//motion row 3, cycle cont / single
ModeRow3	(	iStationNumber		:=1,
				iRowNumber			:=3,
				iAdvanceLimit		:=gHMIButtons.btnFdbk.btn10Fdbk,
				iReturnLimit		:=gHMIButtons.btnFdbk.btn13Fdbk,
				iAdvanceCoil		:=gModeAlternate.gModeButtons.gMotionRow3btn.btnAdvance,
				iReturnCoil			:=gModeAlternate.gModeButtons.gMotionRow3btn.btnReturn,
				iAdvanceTime		:=,
				iReturnTime			:=,
				iAdvanceInterlock	:=,
				iReturnInterlock	:=,
				iAdvancePrompt		:=,
				iReturnPrompt		:=,
				iConfig				:=RowConfig.FullRowNoVal,
				iAdvanceNumber		:=0,
				iReturnNumber		:=0,
				iUnits				:='',
				iPosn				:='',
				NumRows				:=tNumRows,
				MotionRowLocation	:=gModeAlternate.gModeRows.gMotionRow3,
				MotionRowBtnLocation:=gModeAlternate.gModeButtons.gMotionRow3btn
				);
				
//manually set row number for textlist offset				
gModeAlternate.gModeRows.gMotionRow3.IndexLocation := gModeAlternate.gModeRows.gMotionRow3.IndexLocation + 10000;			


//motion row 4, cycle start / stop
ModeRow4	(	iStationNumber		:=1,
				iRowNumber			:=4,
				iAdvanceLimit		:=gHMIButtons.btnFdbk.btnAutoCyclingFdbk,
				iReturnLimit		:=NOT gHMIButtons.btnFdbk.btnAutoCyclingFdbk,
				iAdvanceCoil		:=gModeAlternate.gModeButtons.gMotionRow4btn.btnAdvance,
				iReturnCoil			:=gModeAlternate.gModeButtons.gMotionRow4btn.btnReturn,
				iAdvanceTime		:=,
				iReturnTime			:=,
				iAdvanceInterlock	:=,
				iReturnInterlock	:=,
				iAdvancePrompt		:=,
				iReturnPrompt		:=,
				iConfig				:=RowConfig.FullRowNoVal,
				iAdvanceNumber		:=0,
				iReturnNumber		:=0,
				iUnits				:='',
				iPosn				:='',
				NumRows				:=tNumRows,
				MotionRowLocation	:=gModeAlternate.gModeRows.gMotionRow4,
				MotionRowBtnLocation:=gModeAlternate.gModeButtons.gMotionRow4btn
				);
				
//manually set row number for textlist offset				
gModeAlternate.gModeRows.gMotionRow4.IndexLocation := gModeAlternate.gModeRows.gMotionRow4.IndexLocation + 10000;			

//motion row 5, return home
ModeRow5	(	iStationNumber		:=1,
				iRowNumber			:=5,
				iAdvanceLimit		:=gHMIData.hmiHeader.homestate = 2,
				iReturnLimit		:=gHMIData.hmiHeader.homestate <> 2,
				iAdvanceCoil		:=gModeAlternate.gModeButtons.gMotionRow5btn.btnAdvance,
				iReturnCoil			:=gModeAlternate.gModeButtons.gMotionRow5btn.btnReturn,
				iAdvanceTime		:=,
				iReturnTime			:=,
				iAdvanceInterlock	:=,
				iReturnInterlock	:=,
				iAdvancePrompt		:=,
				iReturnPrompt		:=,
				iConfig				:=RowConfig.OnlyRightNoVal,
				iAdvanceNumber		:=0,
				iReturnNumber		:=0,
				iUnits				:='',
				iPosn				:='',
				NumRows				:=tNumRows,
				MotionRowLocation	:=gModeAlternate.gModeRows.gMotionRow5,
				MotionRowBtnLocation:=gModeAlternate.gModeButtons.gMotionRow5btn
				);
				
//manually set row number for textlist offset				
gModeAlternate.gModeRows.gMotionRow5.IndexLocation := gModeAlternate.gModeRows.gMotionRow5.IndexLocation + 10000;			

//motion row 6, spare
ModeRow6	(	iStationNumber		:=1,
				iRowNumber			:=6,
				iAdvanceLimit		:=FALSE,
				iReturnLimit		:=FALSE,
				iAdvanceCoil		:=gModeAlternate.gModeButtons.gMotionRow6btn.btnAdvance,
				iReturnCoil			:=gModeAlternate.gModeButtons.gMotionRow6btn.btnReturn,
				iAdvanceTime		:=,
				iReturnTime			:=,
				iAdvanceInterlock	:=,
				iReturnInterlock	:=,
				iAdvancePrompt		:=,
				iReturnPrompt		:=,
				iConfig				:=RowConfig.HideAll,
				iAdvanceNumber		:=0,
				iReturnNumber		:=0,
				iUnits				:='',
				iPosn				:='',
				NumRows				:=tNumRows,
				MotionRowLocation	:=gModeAlternate.gModeRows.gMotionRow6,
				MotionRowBtnLocation:=gModeAlternate.gModeButtons.gMotionRow6btn
				);
				
//manually set row number for textlist offset				
gModeAlternate.gModeRows.gMotionRow6.IndexLocation := gModeAlternate.gModeRows.gMotionRow6.IndexLocation + 10000;			

//motion row 7, spare
ModeRow7	(	iStationNumber		:=1,
				iRowNumber			:=7,
				iAdvanceLimit		:=FALSE,
				iReturnLimit		:=FALSE,
				iAdvanceCoil		:=gModeAlternate.gModeButtons.gMotionRow7btn.btnAdvance,
				iReturnCoil			:=gModeAlternate.gModeButtons.gMotionRow7btn.btnReturn,
				iAdvanceTime		:=,
				iReturnTime			:=,
				iAdvanceInterlock	:=,
				iReturnInterlock	:=,
				iAdvancePrompt		:=,
				iReturnPrompt		:=,
				iConfig				:=RowConfig.HideAll,
				iAdvanceNumber		:=0,
				iReturnNumber		:=0,
				iUnits				:='',
				iPosn				:='',
				NumRows				:=tNumRows,
				MotionRowLocation	:=gModeAlternate.gModeRows.gMotionRow7,
				MotionRowBtnLocation:=gModeAlternate.gModeButtons.gMotionRow7btn
				);

//manually set row number for textlist offset				
gModeAlternate.gModeRows.gMotionRow7.IndexLocation := gModeAlternate.gModeRows.gMotionRow7.IndexLocation + 10000;			
				
//motion row 8, gate lock, return only
ModeRow8	(	iStationNumber		:=1,
				iRowNumber			:=8,
				iAdvanceLimit		:=FALSE,
				iReturnLimit		:=gHMIButtons.btnFdbk.btn22Fdbk,
				iAdvanceCoil		:=gModeAlternate.gModeButtons.gMotionRow8btn.btnAdvance,
				iReturnCoil			:=gModeAlternate.gModeButtons.gMotionRow8btn.btnReturn,
				iAdvanceTime		:=,
				iReturnTime			:=,
				iAdvanceInterlock	:=,
				iReturnInterlock	:=,
				iAdvancePrompt		:=,
				iReturnPrompt		:=,
				iConfig				:=RowConfig.OnlyRightNoVal,
				iAdvanceNumber		:=0,
				iReturnNumber		:=0,
				iUnits				:='',
				iPosn				:='',
				NumRows				:=tNumRows,
				MotionRowLocation	:=gModeAlternate.gModeRows.gMotionRow8,
				MotionRowBtnLocation:=gModeAlternate.gModeButtons.gMotionRow8btn
				);
				
//manually set row number for textlist offset				
gModeAlternate.gModeRows.gMotionRow8.IndexLocation := gModeAlternate.gModeRows.gMotionRow8.IndexLocation + 10000;			

//motion row 9, gate unlocks
ModeRow9	(	iStationNumber		:=1,
				iRowNumber			:=9,
				iAdvanceLimit		:=gHMIButtons.btnFdbk.btn20Fdbk,
				iReturnLimit		:=gHMIButtons.btnFdbk.btn21Fdbk,
				iAdvanceCoil		:=gModeAlternate.gModeButtons.gMotionRow9btn.btnAdvance,
				iReturnCoil			:=gModeAlternate.gModeButtons.gMotionRow9btn.btnReturn,
				iAdvanceTime		:=,
				iReturnTime			:=,
				iAdvanceInterlock	:=,
				iReturnInterlock	:=,
				iAdvancePrompt		:=,
				iReturnPrompt		:=,
				iConfig				:=RowConfig.FullRowNoVal,
				iAdvanceNumber		:=0,
				iReturnNumber		:=0,
				iUnits				:='',
				iPosn				:='',
				NumRows				:=tNumRows,
				MotionRowLocation	:=gModeAlternate.gModeRows.gMotionRow9,
				MotionRowBtnLocation:=gModeAlternate.gModeButtons.gMotionRow9btn
				);
				
//manually set row number for textlist offset				
gModeAlternate.gModeRows.gMotionRow9.IndexLocation := gModeAlternate.gModeRows.gMotionRow9.IndexLocation + 10000;
END_ACTION

END_PROGRAM

// ---- HMI1/Screens/Machine Settings/pouMachineSettings.TcPOU
PROGRAM pouMachineSettings
VAR
	btnOSRRead:R_TRIG;
	btnOSRWrite:R_TRIG;
	ii: INT;
	OSRReadLogicDone:R_TRIG;
	
	csvRead:FB_ReadParams;
	csvWrite:FB_WriteParams;
END_VAR

//capture OSR for buttons
btnOSRRead	(	CLK := MachineSettings.btnRead);
btnOSRWrite	(	CLK := MachineSettings.btnWrite);

actReadFile();
actWriteFile();


IF MachineSettings.varSelectedRowValid THEN
		MachineSettings.numSelectedSetting := MachineSettings.Setting[MachineSettings.varSelectedRow].Value;
END_IF

IF MachineSettings.btnMoveValue THEN
	  IF 	MachineSettings.Setting[MachineSettings.varSelectedRow].Value <> MachineSettings.numSelectedSettingNew THEN
			
			//update view
			MachineSettings.Setting[MachineSettings.varSelectedRow].hasChanged := TRUE;
			MachineSettings.Setting[MachineSettings.varSelectedRow].Value := 	MachineSettings.numSelectedSettingNew;
			
			//update data area to write to
			MachineSettings.csvData[MachineSettings.varSelectedRow,1] := INT_TO_STRING (MachineSettings.Setting[MachineSettings.varSelectedRow].Value);
	  END_IF
END_IF


//feedback status
IF csvRead.qStep > 1 THEN
	MachineSettings.strStatusFeeback := 'Reading...';
END_IF
IF csvWrite.qStep > 1 THEN
	MachineSettings.strStatusFeeback := 'Writing...';
END_IF
IF csvRead.qStep = 0 AND csvWrite.qStep = 0 THEN
	MachineSettings.strStatusFeeback := '';
END_IF

IF csvRead.qErrId > 0 THEN
	MachineSettings.strStatusFeeback := CONCAT(STR1:='Read Error ',STR2:=UDINT_TO_STRING(csvRead.qErrId));
END_IF
IF csvWrite.qErrId > 0 THEN
	MachineSettings.strStatusFeeback := CONCAT(STR1:='Write Error ',STR2:=UDINT_TO_STRING(csvWrite.qErrId));
END_IF

ACTION actReadFile:
//read data
csvRead (iRead :=btnOSRRead.Q,
		iNetId :=,
		iFileName:=constCSV.str_mc_filelocation,
		iqdatabase := MachineSettings.csvData
		);

	//check state as output
	OSRReadLogicDone(clk := csvRead.qStep = 0);
	
	
//tidy up HMI screen data
IF OSRReadLogicDone.Q THEN
	MachineSettings.numElementsOfSettings := 0;
	FOR ii:=0 TO 100 DO
		MachineSettings.numElementsOfSettings := ii;
		MachineSettings.Setting[ii].Value := STRING_TO_INT(MachineSettings.csvData[ii,1]);
		MachineSettings.Setting[ii].TextName := MachineSettings.csvData[ii,0];
		MachineSettings.Setting[ii].hasChanged := FALSE;
		IF MachineSettings.csvData[ii,0] = '' THEN
			RETURN;
		END_IF
	END_FOR;
END_IF
END_ACTION

ACTION actWriteFile:
//write data
csvWrite (iWrite :=btnOSRWrite.Q,
		iNetId :=,
		iFileName:=constCSV.str_mc_filelocation,
		iqdatabase := MachineSettings.csvData
		);
		
//tidy up HMI screen data		
IF btnOSRWrite.Q THEN
	FOR ii:=0 TO 100 DO
		MachineSettings.Setting[ii].hasChanged := FALSE;
	END_FOR;
END_IF
END_ACTION

END_PROGRAM

// ---- HMI1/Screens/Machine Settings/FB_ReadParams.TcPOU
FUNCTION_BLOCK FB_ReadParams
VAR_INPUT
	iRead			: BOOL := FALSE;(* Rising edge starts program execution *)
	iNetId			: T_AmsNetId := '';	(* TwinCAT system network address *)
	iFileName		: T_MaxString := '';(* CSV source file path and name *)

END_VAR
VAR_OUTPUT
	qBusy			: BOOL;
	qError			: BOOL;
	qErrId			: UDINT;
	qStep			:DWORD;
END_VAR
VAR
	nRow	 		: UDINT 	:= 0;(* Row number (record) *)
	nColumn			: UDINT 	:= 0;(* Column number (record field) *)
	hFile			: UINT		:= 0;(* File handle of the source file *)
	step			: DWORD 	:= 0;
	fbFileOpen		: FB_FileOpen;(* Opens file *)
	fbFileClose		: FB_FileClose;(* Closes file *)
	fbFileGets		: FB_FileGets;(* Reads one record (line) *)
	fbReader		: FB_CSVMemBufferReader;(* Helper function block used to parse CSV data bytes (single record line) *)
	sCSVLine		: T_MaxString := '';(* Single CSV text line (row, record), we are using string as record buffer (your are able to see read fields)  *)
	sCSVField		: T_MaxString := '';(* Single CSV field value (column, record field) *)


END_VAR

VAR_IN_OUT
		iqdatabase		: ARRAY[0..constCSV.MAX_CSV_ROWS, 0..constCSV.MAX_CSV_COLUMNS ] OF STRING(constCSV.MAX_CSV_FIELD_LENGTH);(* Target PLC database *)
END_VAR

//based on sample code from Beckhoff 35419787.html

CASE step OF
	0:	(* Wait for rising edge at bRead variable *)
		IF iRead THEN
		//	bRead 	:= FALSE;
			qBusy 	:= TRUE;
			qError	:= FALSE;
			qErrId	:= 0;
			hFile	:= 0;
			nRow	:= 0;
			nColumn	:= 0;
			MEMSET( ADR( iqdatabase ), 0, SIZEOF( iqdatabase ) );
			step 		:= 1;
		END_IF

	1:	(* Open source file *)
		fbFileOpen(  bExecute := FALSE  );
		fbFileOpen( sNetId := iNetId, sPathName := iFileName, nMode := FOPEN_MODEREAD OR FOPEN_MODETEXT,(* Open file in TEXT mode! *)
					ePath := PATH_GENERIC, bExecute := TRUE );
		step := 2;

	2:(* Wait until open not busy *)
		fbFileOpen( bExecute := FALSE, bError => qError, nErrID => qErrID, hFile => hFile );
		IF NOT fbFileOpen.bBusy THEN
			IF NOT fbFileOpen.bError THEN
				step := 3;
			ELSE(* Error: file not found? *)
				step := 100;
			END_IF
		END_IF

	3:	(* Read single line (record) *)
		fbFileGets( bExecute := FALSE );
		fbFileGets( sNetId := iNetId, hFile := hFile, bExecute := TRUE );
		step := 4;

	4:(* Wait until read not busy *)
		fbFileGets( bExecute := FALSE, bError => qError, nErrID => qErrID, sLine => sCSVLine );
		IF NOT fbFileGets.bBusy THEN
			IF NOT fbFileGets.bError THEN
				IF fbFileGets.bEOF THEN
					step := 10;(* End of file reached => Close source file *)
				ELSE

					(* FB_FileGets returns text line without the CR (carriage return) character.
					We have to restore the CR character (replace the $L character with $R$L characters) *)
					IF RIGHT( sCSVLine, 1 ) = '$L' THEN
						sCSVLine := REPLACE( sCSVLine, '$R$L', 2, LEN( sCSVLine ) );
					END_IF

					step := 5;
				END_IF
			ELSE(* Error *)
				step := 100;
			END_IF
		END_IF

	5:(* Parse single line (record) *)
		fbReader.eCmd := eEnumCmd_First;(* Read first field value *)
		REPEAT
			fbReader( pBuffer := ADR( sCSVLine ), cbBuffer := SIZEOF( sCSVLine ), getValue => sCSVField );
			IF fbReader.bOk THEN
				fbReader.eCmd := eEnumCmd_Next;(* Read next field value *)

				IF ( nRow <= constCSV.MAX_CSV_ROWS ) THEN
					IF ( nColumn <= constCSV.MAX_CSV_COLUMNS ) THEN
						iqdatabase[nRow, nColumn] := CSVFIELD_TO_STRING( sCSVField, FALSE );(* TODO: Save or use the field value in your application *)
					END_IF
				END_IF

				nColumn := nColumn + 1;(* Increment number of read columns *)
				IF fbReader.bCRLF THEN(* CRLF == TRUE => End of reacord reached *)
					nRow 		:= nRow + 1;(* Increment number of read records *)
					nColumn 	:= 0;(* Reset number of columns *)
				END_IF

			ELSE(* Error: End of record reached or all fields read *)
				step := 3;(* Try to read next line *)
			END_IF
		UNTIL NOT fbReader.bOk
		END_REPEAT

	10:	(* Close source file *)
		fbFileClose( bExecute := FALSE );
		fbFileClose( sNetId := iNetId, hFile := hFile, bExecute := TRUE );
		step := 11;

	11:(* Wait until close not busy *)
		fbFileClose( bExecute := FALSE, bError => qError, nErrID => qErrID );
		IF ( NOT fbFileClose.bBusy ) THEN
			hFile := 0;
			step := 100;
		END_IF

	100: (* Error or ready step => cleanup *)
		IF ( hFile <> 0 ) THEN
			step := 10; (* Close the source file *)
		ELSE
			qBusy := FALSE;
			step := 0;	(* Ready *)
		END_IF

END_CASE


//move to outside world
qStep := step;

END_FUNCTION_BLOCK

// ---- HMI1/Screens/Machine Settings/FB_WriteParams.TcPOU
FUNCTION_BLOCK FB_WriteParams
VAR_INPUT
	iWrite			: BOOL := FALSE;(* Rising edge starts program execution *)
	iNetId			: T_AmsNetId := '';	(* TwinCAT system network address *)
	iFileName		: T_MaxString := '';(* CSV destination file path and name *)
END_VAR
VAR_OUTPUT
	qBusy			: BOOL;
	qError			: BOOL;
	qErrId			: UDINT;
	qStep			: DWORD;
END_VAR
VAR
	sCSVLine		: T_MaxString := '';(* Single CSV text line (row, record), we are using string as record buffer (your are able to see created fields) *)
	sCSVField		: T_MaxString := '';(* Single CSV field value (column, record field) *)
	fbFileOpen		: FB_FileOpen;(* Opens file *)
	fbFileClose		: FB_FileClose;(* Closes file *)
	fbFilePuts		: FB_FilePuts;(* Writes one record (line) *)
	fbWriter		: FB_CSVMemBufferWriter;(* Helper function block used to create CSV data bytes (single record line) *)
	nRow	 		: UDINT 	:= 0;(* Row number (record) *)
	nColumn			: UDINT 	:= 0;(* Column number (record field) *)
	hFile			: UINT		:= 0;(* File handle of the source file *)
	step			: DWORD 	:= 0;
END_VAR

VAR_IN_OUT
	iqdatabase		: ARRAY[0..constCSV.MAX_CSV_ROWS, 0..constCSV.MAX_CSV_COLUMNS ] OF STRING(constCSV.MAX_CSV_FIELD_LENGTH);
END_VAR

//based on sample code from Beckhoff 35419787.html

CASE step OF
	0:	(* Wait for rising edge at bWrite variable *)
		IF iWrite THEN
			//iWrite 	:= FALSE;
			qBusy 	:= TRUE;
			qError	:= FALSE;
			qErrId	:= 0;
			hFile	:= 0;
			nRow	:= 0;
			nColumn	:= 0;
			step 	:= 1;
		END_IF

	1:	(* Open source file *)
		fbFileOpen(  bExecute := FALSE  );
		fbFileOpen( sNetId := iNetId, sPathName := iFileName, nMode := FOPEN_MODEWRITE OR FOPEN_MODETEXT,(* Open file in TEXT mode! *)
					ePath := PATH_GENERIC, bExecute := TRUE );
		step := 2;

	2:(* Wait until open not busy *)
		fbFileOpen( bExecute := FALSE, bError => qError, nErrID => qErrId, hFile => hFile );
		IF NOT fbFileOpen.bBusy THEN
			IF NOT fbFileOpen.bError THEN
				step := 3;
			ELSE(* Error: file not found? *)
				step := 100;
			END_IF
		END_IF

	3:(* Convert one PLC record to CSV format *)
		sCSVLine := '';
		fbWriter.eCmd := eEnumCmd_First;(* Write first field value *)
		IF nRow <= constCSV.MAX_CSV_ROWS THEN

			FOR nColumn := 0 TO constCSV.MAX_CSV_COLUMNS BY 1 DO

				sCSVField := STRING_TO_CSVFIELD( iqdatabase[ nRow, nColumn ], FALSE );(* TODO: Get field value from your application *)

				(* Add new field to the record buffer *)
				fbWriter( 	pBuffer := ADR( sCSVLine ), cbBuffer := SIZEOF( sCSVLine ) - 1, putValue := sCSVField, pValue := 0, cbValue := 0,
							bCRLF := ( nColumn = constCSV.MAX_CSV_COLUMNS ) );(* bCRLF == TRUE => Write CRLF after the last field value *)
				IF fbWriter.bOk THEN
					fbWriter.eCmd := eEnumCmd_Next;(* Write next field value *)
				ELSE(* Error *)
					step := 100;
					RETURN;
				END_IF

			END_FOR(* FOR nColumn := 0... *)

			(* FB_FilePuts adds allready CR (carriage return) to the written line.
			We have to replace the $R$L characters with $L character to avoid double CR. *)
			IF RIGHT( sCSVLine, 2 ) = '$R$L' THEN
				sCSVLine := REPLACE( sCSVLine, '$L', 2, LEN( sCSVLine ) - 1 );
			END_IF

			nRow := nRow + 1;(* Increment number of created records (rows) *)
			step := 4;(* Write record to the file *)

		ELSE(* All rows written => Close file *)
			step := 10;
		END_IF

	4:	(* Write single text line *)
		fbFilePuts( bExecute := FALSE );
		fbFilePuts( sNetId := iNetId, hFile := hFile, sLine := sCSVLine, bExecute := TRUE );
		step := 5;

	5:(* Wait until write not busy *)
		fbFilePuts( bExecute := FALSE, bError => qError, nErrID => qErrId );
		IF NOT fbFilePuts.bBusy THEN
			IF NOT fbFilePuts.bError THEN
				step := 3;(* Write next record *)
			ELSE(* Error *)
				step := 100;
			END_IF
		END_IF

	10:	(* Close source file *)
		fbFileClose( bExecute := FALSE );
		fbFileClose( sNetId := iNetId, hFile := hFile, bExecute := TRUE );
		step := 11;

	11:(* Wait until close not busy *)
		fbFileClose( bExecute := FALSE, bError => qError, nErrID => qErrId );
		IF ( NOT fbFileClose.bBusy ) THEN
			hFile := 0;
			step := 100;
		END_IF

	100: (* Error or ready step => cleanup *)
		IF ( hFile <> 0 ) THEN
			step := 10; (* Close the source file *)
		ELSE
			qBusy := FALSE;
			step := 0;	(* Ready *)
		END_IF

END_CASE


//move to outside world
qStep := step;

END_FUNCTION_BLOCK

// ---- Data Collection/dataAnalyse/prgDataAnaylse.TcPOU
PROGRAM prgDataAnaylse
VAR
	windowCheck:FB_Window;
	
END_VAR

//windowCheck	(dataAxis := dataGrab.	,
//			);

END_PROGRAM

// ---- HMI1/Logic/FC_Setup.TcPOU
FUNCTION FC_Setup : bool
VAR_INPUT
END_VAR
VAR
END_VAR

//READ ME FIRST////////////////////////////
///////////////////////////////////////////
//For a given machine, enable the stationEnables below for the presence of a station
//If a stationEnable is FALSE, then the related allowX below are not used

(*
General Setup Instructions
1. Follow this FC_Setup and set values TRUE/FALSE as required. Typically, only the .stationEnables can be set
2. Define the motions in the system by editing the 'MotionRowText' text list.
3. Add IO mapping and motion name text to fault messages in the system by editing the textlists in the 'X_Language Text' folder.
4. Add Power on logic
5. Add interlocks for each motion in "Sx_xx_Motion_xx_xx" PRGs in "MyAdvanceInterlock" and "MyReturnInterlock"
6. Map Inputs and outputs using "Sx_IO.Rowxx.qAdvanceCoil/Sx_IO.Rowxx.qReturnedCoil" and "Sxx_IO.Rowxx.iAdvanceDepth/Sx_IO.Rowxx.iReturnedDepth"
7. Test each motion using manual mode. Each device, e.g. a cylinder should advance and return
8. Edit other FB_HMI_Control values as required
9. Add auto logic
10. Auto Cycle --> Start
*)

//station names
//open the text list "StationNames" and edit

//setup machine
System.gSetup.stationEnable[1] := TRUE; //TRUE if station is present
System.gSetup.stationEnable[2] := FALSE; //FALSE if the station does not exist on this machine
System.gSetup.stationEnable[3] := FALSE;
System.gSetup.stationEnable[4] := FALSE;
System.gSetup.stationEnable[5] := FALSE;
System.gSetup.stationEnable[6] := FALSE;

//number of rows in each station
System.gSetup.stationFunctions[1].numRowsConfig := 9;		//18 is two pages
System.gSetup.stationFunctions[2].numRowsConfig := 9;		//9 is one page
System.gSetup.stationFunctions[3].numRowsConfig := 99;		//up to 99 rows
System.gSetup.stationFunctions[4].numRowsConfig := 99;
System.gSetup.stationFunctions[5].numRowsConfig := 99;
System.gSetup.stationFunctions[6].numRowsConfig := 99;

//set up cycle time setpoints
S1_Global.station.part.CycleTimeTarget := 60;
S1_Global.station.part.CycleTimeGrossOver := S1_Global.station.part.CycleTimeTarget  * 2;

S2_Global.station.part.CycleTimeTarget := 60;
S2_Global.station.part.CycleTimeGrossOver := S2_Global.station.part.CycleTimeTarget  * 2;

S3_Global.station.part.CycleTimeTarget := 60;
S3_Global.station.part.CycleTimeGrossOver := S3_Global.station.part.CycleTimeTarget  * 2;

S4_Global.station.part.CycleTimeTarget := 60;
S4_Global.station.part.CycleTimeGrossOver := S4_Global.station.part.CycleTimeTarget  * 2;

S5_Global.station.part.CycleTimeTarget := 60;
S5_Global.station.part.CycleTimeGrossOver := S5_Global.station.part.CycleTimeTarget  * 2;

S6_Global.station.part.CycleTimeTarget := 60;
S6_Global.station.part.CycleTimeGrossOver := S6_Global.station.part.CycleTimeTarget  * 2;

//station features
System.gSetup.stationFunctions[1].allowAutoCycle := TRUE;	//TRUE to allow auto cycle
System.gSetup.stationFunctions[1].allowManualMode := TRUE;	//Generally speaking....
System.gSetup.stationFunctions[1].allowSemiAuto := TRUE; 	//..all functions are enabled...
System.gSetup.stationFunctions[1].allowDryCycle := TRUE;	//..unless there is a good reason...
System.gSetup.stationFunctions[1].allowBypass := TRUE;		//..to disable them.
System.gSetup.stationFunctions[1].allowContinuousCycle := TRUE;
System.gSetup.stationFunctions[1].allowSingleCycle := TRUE;
System.gSetup.stationFunctions[1].allowSEOC := TRUE;
System.gSetup.stationFunctions[1].allowPowerOn := TRUE;
System.gSetup.stationFunctions[1].allowPowerOff := TRUE;
System.gSetup.stationFunctions[1].allowServicesPowerOn := TRUE;
System.gSetup.stationFunctions[1].allowRemoteControl := TRUE;
System.gSetup.stationFunctions[1].allowServicesPowerOn := TRUE;
System.gSetup.stationFunctions[1].allowSilenceHorn := TRUE;
System.gSetup.stationFunctions[1].allowGate1Req := TRUE;
System.gSetup.stationFunctions[1].allowGate2Req := TRUE;
System.gSetup.stationFunctions[1].allowLockAccessGates := TRUE;
System.gSetup.stationFunctions[1].allowEnablePendent := TRUE;


System.gSetup.stationFunctions[2].allowAutoCycle := TRUE;
System.gSetup.stationFunctions[2].allowManualMode := TRUE;
System.gSetup.stationFunctions[2].allowSemiAuto := TRUE;
System.gSetup.stationFunctions[2].allowDryCycle := TRUE;
System.gSetup.stationFunctions[2].allowBypass := TRUE;
System.gSetup.stationFunctions[2].allowContinuousCycle := TRUE;
System.gSetup.stationFunctions[2].allowSingleCycle := TRUE;
System.gSetup.stationFunctions[2].allowSEOC := TRUE;
System.gSetup.stationFunctions[2].allowPowerOn := TRUE;
System.gSetup.stationFunctions[2].allowPowerOff := TRUE;
System.gSetup.stationFunctions[2].allowServicesPowerOn := TRUE;
System.gSetup.stationFunctions[2].allowRemoteControl := TRUE;
System.gSetup.stationFunctions[2].allowServicesPowerOn := TRUE;
System.gSetup.stationFunctions[2].allowSilenceHorn := TRUE;
System.gSetup.stationFunctions[2].allowGate1Req := TRUE;
System.gSetup.stationFunctions[2].allowGate2Req := TRUE;
System.gSetup.stationFunctions[2].allowLockAccessGates := TRUE;
System.gSetup.stationFunctions[2].allowEnablePendent := TRUE;

System.gSetup.stationFunctions[3].allowAutoCycle := TRUE;
System.gSetup.stationFunctions[3].allowManualMode := TRUE;
System.gSetup.stationFunctions[3].allowSemiAuto := TRUE;
System.gSetup.stationFunctions[3].allowDryCycle := TRUE;
System.gSetup.stationFunctions[3].allowBypass := TRUE;
System.gSetup.stationFunctions[3].allowContinuousCycle := TRUE;
System.gSetup.stationFunctions[3].allowSingleCycle := TRUE;
System.gSetup.stationFunctions[3].allowSEOC := TRUE;
System.gSetup.stationFunctions[3].allowPowerOn := TRUE;
System.gSetup.stationFunctions[3].allowPowerOff := TRUE;
System.gSetup.stationFunctions[3].allowServicesPowerOn := TRUE;
System.gSetup.stationFunctions[3].allowRemoteControl := TRUE;
System.gSetup.stationFunctions[3].allowServicesPowerOn := TRUE;
System.gSetup.stationFunctions[3].allowSilenceHorn := TRUE;
System.gSetup.stationFunctions[3].allowGate1Req := TRUE;
System.gSetup.stationFunctions[3].allowGate2Req := TRUE;
System.gSetup.stationFunctions[3].allowLockAccessGates := TRUE;
System.gSetup.stationFunctions[3].allowEnablePendent := TRUE;

System.gSetup.stationFunctions[4].allowAutoCycle := TRUE;
System.gSetup.stationFunctions[4].allowManualMode := TRUE;
System.gSetup.stationFunctions[4].allowSemiAuto := TRUE;
System.gSetup.stationFunctions[4].allowDryCycle := TRUE;
System.gSetup.stationFunctions[4].allowBypass := TRUE;
System.gSetup.stationFunctions[4].allowContinuousCycle := TRUE;
System.gSetup.stationFunctions[4].allowSingleCycle := TRUE;
System.gSetup.stationFunctions[4].allowSEOC := TRUE;
System.gSetup.stationFunctions[4].allowPowerOn := TRUE;
System.gSetup.stationFunctions[4].allowPowerOff := TRUE;
System.gSetup.stationFunctions[4].allowServicesPowerOn := TRUE;
System.gSetup.stationFunctions[4].allowRemoteControl := TRUE;
System.gSetup.stationFunctions[4].allowServicesPowerOn := TRUE;
System.gSetup.stationFunctions[4].allowSilenceHorn := TRUE;
System.gSetup.stationFunctions[4].allowGate1Req := TRUE;
System.gSetup.stationFunctions[4].allowGate2Req := TRUE;
System.gSetup.stationFunctions[4].allowLockAccessGates := TRUE;
System.gSetup.stationFunctions[4].allowEnablePendent := TRUE;

System.gSetup.stationFunctions[5].allowAutoCycle := TRUE;
System.gSetup.stationFunctions[5].allowManualMode := TRUE;
System.gSetup.stationFunctions[5].allowSemiAuto := TRUE;
System.gSetup.stationFunctions[5].allowDryCycle := TRUE;
System.gSetup.stationFunctions[5].allowBypass := TRUE;
System.gSetup.stationFunctions[5].allowContinuousCycle := TRUE;
System.gSetup.stationFunctions[5].allowSingleCycle := TRUE;
System.gSetup.stationFunctions[5].allowSEOC := TRUE;
System.gSetup.stationFunctions[5].allowPowerOn := TRUE;
System.gSetup.stationFunctions[5].allowPowerOff := TRUE;
System.gSetup.stationFunctions[5].allowServicesPowerOn := TRUE;
System.gSetup.stationFunctions[5].allowRemoteControl := TRUE;
System.gSetup.stationFunctions[5].allowServicesPowerOn := TRUE;
System.gSetup.stationFunctions[5].allowSilenceHorn := TRUE;
System.gSetup.stationFunctions[5].allowGate1Req := TRUE;
System.gSetup.stationFunctions[5].allowGate2Req := TRUE;
System.gSetup.stationFunctions[5].allowLockAccessGates := TRUE;
System.gSetup.stationFunctions[5].allowEnablePendent := TRUE;

System.gSetup.stationFunctions[6].allowAutoCycle := TRUE;
System.gSetup.stationFunctions[6].allowManualMode := TRUE;
System.gSetup.stationFunctions[6].allowSemiAuto := TRUE;
System.gSetup.stationFunctions[6].allowDryCycle := TRUE;
System.gSetup.stationFunctions[6].allowBypass := TRUE;
System.gSetup.stationFunctions[6].allowContinuousCycle := TRUE;
System.gSetup.stationFunctions[6].allowSingleCycle := TRUE;
System.gSetup.stationFunctions[6].allowSEOC := TRUE;
System.gSetup.stationFunctions[6].allowPowerOn := TRUE;
System.gSetup.stationFunctions[6].allowPowerOff := TRUE;
System.gSetup.stationFunctions[6].allowServicesPowerOn := TRUE;
System.gSetup.stationFunctions[6].allowRemoteControl := TRUE;
System.gSetup.stationFunctions[6].allowServicesPowerOn := TRUE;
System.gSetup.stationFunctions[6].allowSilenceHorn := TRUE;
System.gSetup.stationFunctions[6].allowGate1Req := TRUE;
System.gSetup.stationFunctions[6].allowGate2Req := TRUE;
System.gSetup.stationFunctions[6].allowLockAccessGates := TRUE;
System.gSetup.stationFunctions[6].allowEnablePendent := TRUE;

//latch XIC messages?
S1_Global.station.Data.latchXICmsg := TRUE;
S2_Global.station.Data.latchXICmsg := FALSE;
S3_Global.station.Data.latchXICmsg := FALSE;
S4_Global.station.Data.latchXICmsg := FALSE;
S5_Global.station.Data.latchXICmsg := FALSE;
S6_Global.station.Data.latchXICmsg := FALSE;

END_FUNCTION

// ---- HMI1/Logic/VisuInit.TcPOU
PROGRAM VisuInit
VAR
END_VAR

gHMIData.gVisuHasInited := TRUE;

END_PROGRAM

// ---- Project Information/F_GetCompany.TcPOU
// This function has been automatically generated from the project information.
{attribute 'signature_flag' := '1073741824'}
{attribute 'TcGenerated'}
{attribute 'no-analysis'}
FUNCTION F_GetCompany : WSTRING
VAR_INPUT
	
END_VAR

F_GetCompany := "Company Name";

END_FUNCTION

// ---- Project Information/F_GetTitle.TcPOU
// This function has been automatically generated from the project information.
{attribute 'signature_flag' := '1073741824'}
{attribute 'TcGenerated'}
{attribute 'no-analysis'}
FUNCTION F_GetTitle : WSTRING
VAR_INPUT
	
END_VAR

F_GetTitle := "Project Title";

END_FUNCTION

// ---- Project Information/F_GetVersion.TcPOU
// This function has been automatically generated from the project information.
{attribute 'signature_flag' := '1073741824'}
{attribute 'TcGenerated'}
{attribute 'no-analysis'}
FUNCTION F_GetVersion : ST_LibVersion
VAR_INPUT
	
END_VAR

F_GetVersion.iMajor := 0;
F_GetVersion.iMinor := 0;
F_GetVersion.iBuild := 1;
F_GetVersion.iRevision := 1;
F_GetVersion.sVersion := '0.0.1.1';
F_GetVersion.nFlags := 0;

END_FUNCTION

// ---- X_Sim/FB_SimMotion.TcPOU
FUNCTION_BLOCK FB_SimMotion
VAR_INPUT
	iAdvanceReq:BOOL;
	iReturnReq:BOOL;
	iClear:BOOL;
	
END_VAR

VAR_OUTPUT
	qAdvanced:BOOL;
	qReturned:BOOL;
END_VAR
VAR
	timAdvanceDelay: TON;
	timReturnDelay: TON;
END_VAR

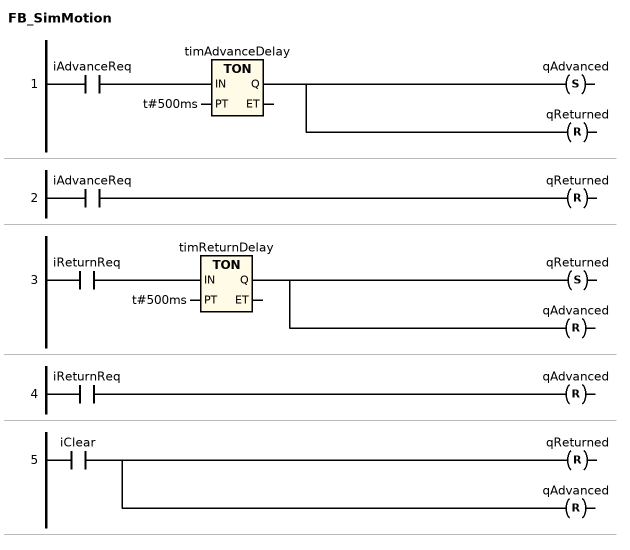
// NETWORK 1
timAdvanceDelay(IN := iAdvanceReq, PT := t#500ms); // TON
qAdvanced S= timAdvanceDelay.Q;
qReturned R= timAdvanceDelay.Q;

// NETWORK 2
qReturned R= iAdvanceReq;

// NETWORK 3
timReturnDelay(IN := iReturnReq, PT := t#500ms); // TON
qReturned S= timReturnDelay.Q;
qAdvanced R= timReturnDelay.Q;

// NETWORK 4
qAdvanced R= iReturnReq;

// NETWORK 5
qReturned R= iClear;
qAdvanced R= iClear;

END_FUNCTION_BLOCK

// ---- Data Collection/Dat_550_DataAxis.TcVIS
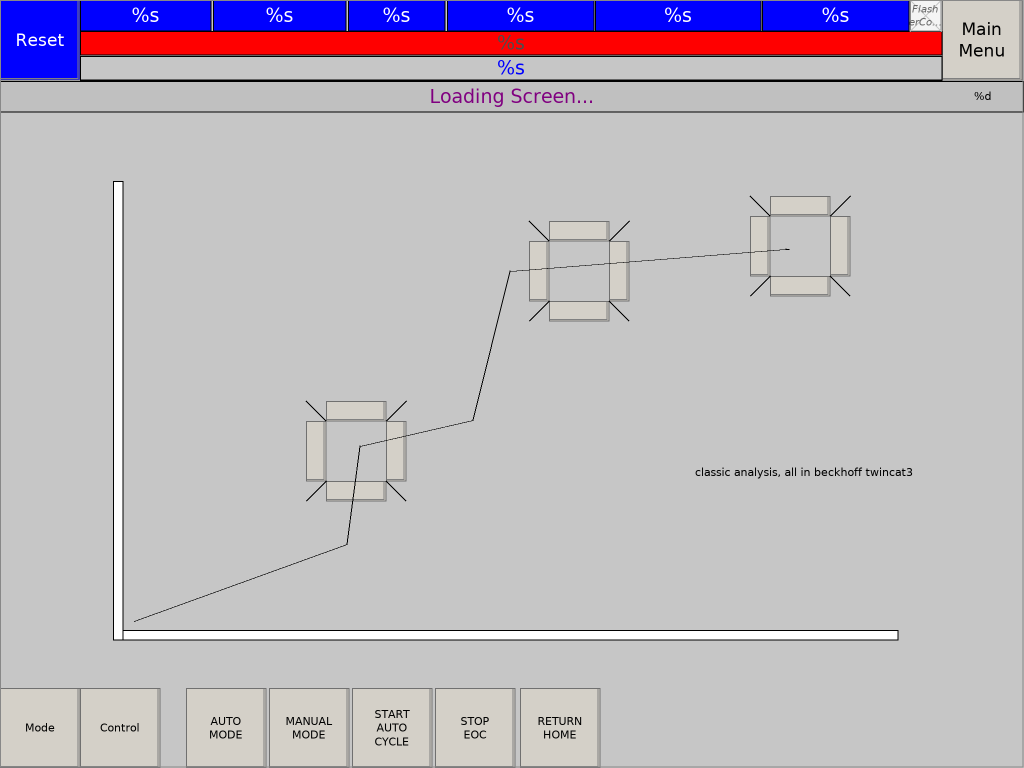
VISUALIZATION Dat_550_DataAxis  // 1024x768
    Frame (0,0 1024x768)
        shows Tmp_000_Template(header := gHMIData.hmiHeader)
    Frame (306,401 100x100)
        shows diaDataBox(iqBoxdata := dataGrab.dataCurrentVisu.box1)
    Frame (529,221 100x100)
        shows diaDataBox(iqBoxdata := dataGrab.dataCurrentVisu.box2)
    Frame (750,196 100x100)
        shows diaDataBox(iqBoxdata := dataGrab.dataCurrentVisu.box3)
    Rectangle (113,630 785x10)
    Rectangle (113,181 10x459)
    Polyline (134,621) (347,544) (360,446) (473,420) (510,271) (786,249) (789,249)
    Label (667,461 274x23), "classic analysis, all in beckhoff twincat3"
END_VISUALIZATION

// ---- Data Collection/dynamicBox/diaDataBox.TcVIS
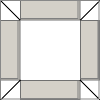
VISUALIZATION diaDataBox  // 100x100
VAR_IN_OUT
	iqBoxdata:structBoxData;
	
END_VAR
    Button (20,0 60x20), text list: 'textListTop', text index: iqBoxdata.topStatus.EntryRule
        OnMouseClick: toggle iqBoxdata.topStatusChange
    Button (0,20 20x60), text list: 'textListLeft', text index: iqBoxdata.leftStatus.EntryRule
        OnMouseClick: toggle iqBoxdata.leftStatusChange
    Button (80,20 20x60), text list: 'textListRight', text index: iqBoxdata.rightStatus.EntryRule
        OnMouseClick: toggle iqBoxdata.rightStatusChange
    Button (20,80 60x20), text list: 'textListBottom', text index: iqBoxdata.bottomStatus.EntryRule
        OnMouseClick: toggle iqBoxdata.bottomStatusChange
    Line (20,20) (0,0)
    Line (100,100) (80,80)
    Line (100,0) (80,20)
    Line (20,80) (0,100)
END_VISUALIZATION

// ---- Data Collection/dynamicBox/textListLeft.TcTLO
TEXTLIST textListLeft
  0 = ''
  1 = 'X'
  2 = '>'
  3 = '<'
   = ''
END_TEXTLIST

// ---- Data Collection/dynamicBox/textListRight.TcTLO
TEXTLIST textListRight
  0 = ''
  1 = 'X'
  2 = '>'
  3 = '<'
   = ''
END_TEXTLIST

// ---- Data Collection/dynamicBox/textListTop.TcTLO
TEXTLIST textListTop
  0 = ''
  1 = 'X'
  2 = 'V '
  3 = 'Λ'
   = ''
END_TEXTLIST

// ---- Data Collection/dynamicBox/textListBottom.TcTLO
TEXTLIST textListBottom
  0 = ''
  1 = 'X'
  2 = 'Λ'
  3 = 'V'
   = ''
END_TEXTLIST

// ---- HMI1/Data/ManualPageTitle.TcTLO
TEXTLIST ManualPageTitle
  10001 = '==Line1=OP0010' | 汉语: '汉语'
  10005 = 'Page 5 s1'
  10004 = 'Page 4 s1'
  10003 = 'Page 3 s1'
  10002 = 'Page 2 s1'
  10006 = 'Page 6 s1'
  20001 = 'Page 1 s2'
  20002 = 'Page 2 s2'
  20003 = 'Page 3 s2'
  20004 = 'Page 4 s2'
  20005 = 'Page 5 s2'
  20006 = 'Page 6 s2'
  30001 = 'Page 1 s3'
  30002 = 'Page 2 s3'
  30003 = 'Page 3 s3'
  30004 = 'Page 4 s3'
  30005 = 'Page 5 s3'
  30006 = 'Page 6 s3'
  40001 = 'Page 1 s4'
  40002 = 'Page 2 s4'
  40003 = 'Page 3 s4'
  40004 = 'Page 4 s4'
  40005 = 'Page 5 s4'
  40006 = 'Page 6 s4'
  50001 = 'Page 1 s5'
  50002 = 'Page 2 s5'
  50003 = 'Page 3 s5'
  50004 = 'Page 4 s5'
  50005 = 'Page 5 s5'
  50006 = 'Page 6 s5'
  60001 = 'Page 1 s6'
  60002 = 'Page 2 s6'
  60003 = 'Page 3 s6'
  60004 = 'Page 4 s6'
  60005 = 'Page 5 s6'
  60006 = 'Page 6 s6'
  10007 = 'Page 7 s1'
  10008 = 'Page 8 s1'
  10009 = 'Page 9 s1'
  10010 = 'Page 10 s1'
  10011 = 'Page 11 s1'
   = ''
END_TEXTLIST

// ---- HMI1/Data/ModeRowText.TcTLO
TEXTLIST ModeRowText
  10000 = 'Power On' | 汉语: '汉语'
  10001 = 'Power On' | 汉语: '汉语'
  10002 = '10002' | 汉语: '汉语'
  10003 = 'Power Off' | 汉语: '汉语'
  10004 = 'Power Off' | 汉语: '汉语'
  10005 = '10005'
  10006 = 'Power'
  10007 = '10007'
  10008 = '10008'
  10009 = '10009'
  10010 = '10010'
  10011 = '10011'
  10012 = '10012'
  10013 = '10013'
  10014 = '10014'
  10015 = '10015'
  10016 = '10016'
  10017 = '10017'
  10018 = '10018'
  10019 = '10019'
  10020 = 'Automatic'
  10021 = 'Automatic'
  10022 = '10022'
  10023 = 'Manual'
  10024 = 'Manual'
  10025 = '10025'
  10026 = 'Mode'
  10027 = '10027'
  10028 = '10028'
  10029 = '10029'
  10030 = '10030'
  10031 = '10031'
  10032 = '10032'
  10033 = '10033'
  10034 = '10034'
  10035 = '10035'
  10036 = '10036'
  10037 = '10037'
  10038 = '10038'
  10039 = '10039'
  10040 = 'Continuous Cycle'
  10041 = 'Continuous Cycle'
  10042 = '10042'
  10043 = 'Single Cycle'
  10044 = 'Single Cycle'
  10045 = '10045'
  10046 = 'Cycle'
  10047 = '10047'
  10048 = '10048'
  10049 = '10049'
  10050 = '10050'
  10051 = '10051'
  10052 = '10052'
  10053 = '10053'
  10054 = '10054'
  10055 = '10055'
  10056 = '10056'
  10057 = '10057'
  10058 = '10058'
  10059 = '10059'
  10060 = 'Auto Cycle Start'
  10061 = 'Auto Cycling'
  10062 = '10062'
  10063 = 'Stop Cycle'
  10064 = 'Auto Cycle Stopped'
  10065 = '10065'
  10066 = 'Cycle Start'
  10067 = '10067'
  10068 = '10068'
  10069 = '10069'
  10070 = '10070'
  10071 = '10071'
  10072 = '10072'
  10073 = '10073'
  10074 = '10074'
  10075 = '10075'
  10076 = '10076'
  10077 = '10077'
  10078 = '10078'
  10079 = '10079'
  10080 = '10080'
  10081 = '10081'
  10082 = '10082'
  10083 = 'Return Home'
  10084 = 'Home'
  10085 = '10085'
  10086 = 'Home'
  10087 = '10087'
  10088 = '10088'
  10089 = '10089'
  10090 = '10090'
  10091 = '10091'
  10092 = '10092'
  10093 = '10093'
  10094 = '10094'
  10095 = '10095'
  10096 = '10096'
  10097 = '10097'
  10098 = '10098'
  10099 = '10099'
  10100 = 'To Wash Posn'
  10101 = 'At Wash Posn'
  10102 = '10102'
  10103 = 'To Place Pounce'
  10104 = 'At Place Pounce'
  10105 = '10105'
  10106 = 'Robot'
  10107 = '10107'
  10108 = '10108'
  10109 = '10109'
  10110 = '10110'
  10111 = '10111'
  10112 = '10112'
  10113 = '10113'
  10114 = '10114'
  10115 = '10115'
  10116 = '10116'
  10117 = '10117'
  10118 = '10118'
  10119 = '10119'
  10120 = 'Start Washer'
  10121 = 'Washer On'
  10122 = '10122'
  10123 = 'Stop Washer'
  10124 = 'Washer Off'
  10125 = '10125'
  10126 = 'Washer Jets'
  10127 = '10127'
  10128 = '10128'
  10129 = '10129'
  10130 = '10130'
  10131 = '10131'
  10132 = '10132'
  10133 = '10133'
  10134 = '10134'
  10135 = '10135'
  10136 = '10136'
  10137 = '10137'
  10138 = '10138'
  10139 = '10139'
  10140 = '10140'
  10141 = '10141'
  10142 = '10142'
  10143 = 'Lock'
  10144 = 'Locked'
  10145 = '10145'
  10146 = 'Access Door'
  10147 = '10147'
  10148 = '10148'
  10149 = '10149'
  10150 = '10150'
  10151 = '10151'
  10152 = '10152'
  10153 = '10153'
  10154 = '10154'
  10155 = '10155'
  10156 = '10156'
  10157 = '10157'
  10158 = '10158'
  10159 = '10159'
  10160 = 'Request Access Gate 1'
  10161 = 'Request Access Gate 1'
  10162 = '10162'
  10163 = 'Request Access Gate 2'
  10164 = 'Request Access Gate 2'
  10165 = '10165'
  10166 = 'Access Door'
  10167 = '10167'
  10168 = '10168'
  10169 = '10169'
  10170 = '10170'
  10171 = '10171'
  10172 = '10172'
  10173 = '10173'
  10174 = '10174'
  10175 = '10175'
  10176 = '10176'
  10177 = '10177'
  10178 = '10178'
  10179 = '10179'
  10180 = '10180'
  10181 = '10181'
  10182 = '10182'
  10183 = '10183'
  10184 = '10184'
  10185 = '10185'
  10186 = '10186'
  10187 = '10187'
  10188 = '10188'
  10189 = '10189'
  10190 = '10190'
  10191 = '10191'
  10192 = '10192'
  10193 = '10193'
  10194 = '10194'
  10195 = '10195'
  10196 = '10196'
  10197 = '10197'
  10198 = '10198'
  10199 = '10199'
   = ''
END_TEXTLIST

// ---- HMI1/Data/ScreenNames.TcTLO
TEXTLIST ScreenNames
  801 = 'EtherCAT Diagnostics' | 汉语: '汉语'
  802 = 'PROFIBUS Diagnostics' | 汉语: '汉语'
  803 = 'PROFINET Diagnostics' | 汉语: '汉语'
  800 = 'I/O Memory Display'
  40 = 'Machine Layout'
  30 = 'Menu Screen 1'
  31 = 'Menu Screen 2'
  32 = 'Menu Screen 3'
  20 = 'Alarms'
  21 = 'Alarm View'
  1 = 'Mode Screen'
  10 = 'Motions'
  500 = 'Part Screen'
  900 = 'About'
  901 = 'HMI Screen'
  401 = 'Machine Units'
  402 = 'Axis Screen'
  403 = 'Language Screen'
  32767 = 'No Screen Detected'
  501 = 'Cycle Time'
  11 = 'Axis Data'
  700 = 'Safety Status'
  701 = 'Safety Checksum'
  2 = 'Mode Screen Rows'
   = ''
END_TEXTLIST

// ---- HMI1/Data/stationLinked.TcTLO
TEXTLIST stationLinked
  0 = 'Unlinked'
  1 = 'Linked'
   = ''
END_TEXTLIST

// ---- HMI1/Data/TaskText.TcTLO
TEXTLIST TaskText
  0 = 'No Text' | 汉语: '汉语'
  1 = 'Not Started' | 汉语: '汉语'
  2 = 'Started' | 汉语: '汉语'
  3 = 'Completed'
  4 = 'Passed'
  5 = 'Failed'
  6 = 'Rejected'
  7 = 'Skipped'
  8 = 'Bypassed'
  9 = 'Unknown'
   = ''
END_TEXTLIST

// ---- HMI1/Screens/Diagnostic IO View/Dia_800_DataDisplay.TcVIS
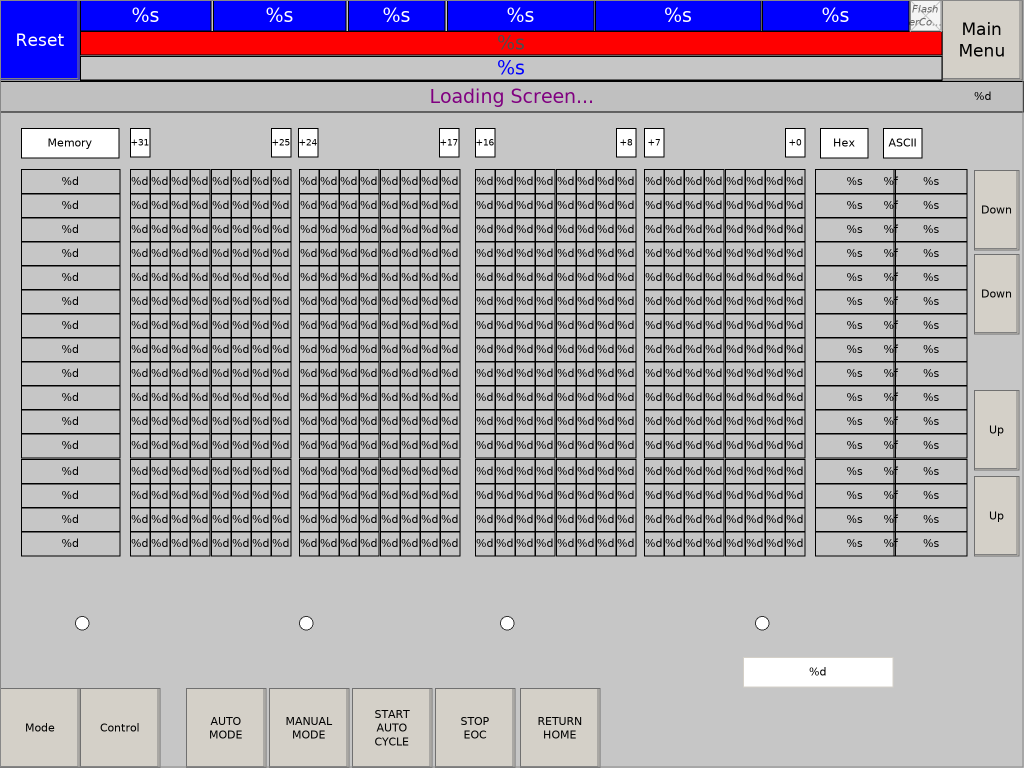
VISUALIZATION Dia_800_DataDisplay  // 1024x768
    Frame (0,0 1024x768)
        shows Tmp_000_Template(header := gHMIData.hmiHeader)
    Frame (21,169 910x26)
        shows visuDataDisplay(d := ioview.ByteRow[0])
        shows visuDataDisplay()
    Frame (21,193 910x26)
        shows visuDataDisplay(d := ioview.ByteRow[1])
    Frame (21,217 910x26)
        shows visuDataDisplay(d := ioview.ByteRow[2])
    Frame (21,241 910x26)
        shows visuDataDisplay(d := ioview.ByteRow[3])
    Frame (21,265 910x26)
        shows visuDataDisplay(d := ioview.ByteRow[4])
    Frame (21,289 910x26)
        shows visuDataDisplay(d := ioview.ByteRow[5])
    Frame (21,313 910x26)
        shows visuDataDisplay(d := ioview.ByteRow[6])
    Frame (21,337 910x26)
        shows visuDataDisplay(d := ioview.ByteRow[7])
    Frame (21,361 910x26)
        shows visuDataDisplay(d := ioview.ByteRow[8])
    Frame (21,385 910x26)
        shows visuDataDisplay(d := ioview.ByteRow[9])
    Frame (21,409 910x26)
        shows visuDataDisplay(d := ioview.ByteRow[10])
    Frame (21,433 910x26)
        shows visuDataDisplay(d := ioview.ByteRow[11])
    Rectangle (21,128 98x30), "Memory"
    Rectangle (883,128 39x30), "ASCII"
    Rectangle (820,128 48x30), "Hex"
    Rectangle (785,128 20x29), "+0"
    Rectangle (644,128 20x29), "+7"
    Rectangle (475,128 20x29), "+16"
    Rectangle (616,128 20x29), "+8"
    Rectangle (439,128 20x29), "+17"
    Rectangle (298,128 20x29), "+24"
    Rectangle (271,128 20x29), "+25"
    Rectangle (130,128 20x29), "+31"
    Frame (21,459 910x26)
        shows visuDataDisplay(d := ioview.ByteRow[12])
    Frame (21,483 910x26)
        shows visuDataDisplay(d := ioview.ByteRow[13])
    Frame (21,507 910x26)
        shows visuDataDisplay(d := ioview.ByteRow[14])
    Frame (21,531 910x26)
        shows visuDataDisplay(d := ioview.ByteRow[15])
    Button (974,476 45x80), "Up"
        tap ioView.btnRaiseFaster
    Button (974,390 45x80), "Up"
        tap ioView.btnRaise
    Button (974,254 45x80), "Down"
        tap ioView.btnLower
    Button (974,170 45x80), "Down"
        tap ioView.btnLowerFaster
    RadioButton (753,583 150x80), variable: ioView.memtype
    RadioButton (73,583 150x80), variable: ioView.memsize
    RadioButton (297,583 230x80), variable: ioView.memHexDisplay
        p340057476: HEX/DEC
    RadioButton (498,583 235x80), variable: ioView.memswap
        p2481256679: SIEMENS/754
    Textfield (743,657 150x30), "%d", text variable: ioView.memoffset
        OnMouseClick: write ioView.memoffset via VisuDialogs.Numpad
END_VISUALIZATION

// ---- HMI1/Screens/Dialogs/dialogEnterValueInteger.TcVIS
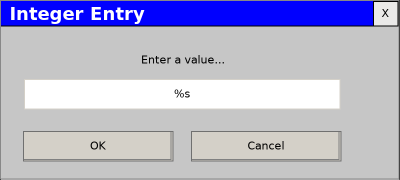
VISUALIZATION dialogEnterValueInteger  // 400x180
VAR_IN_OUT
	enteredValue:INT;
END_VAR
    Rectangle (0,0 400x188)
    Rectangle (0,0 400x26), "Integer Entry"
    Rectangle (373,1 25x25), "X"
        OnMouseClick: CloseDialog Dialog=dialogEnterValueInteger, Result=Cancel, NumpadKeypadSet=True
    Label (108,45 150x30), "Enter a value..."
    Textfield (24,79 316x30), "%s", text variable: enteredValue
        OnMouseClick: write enteredValue via VisuDialogs.Numpad
    Button (23,131 150x30), "OK"
        OnMouseClick: CloseDialog Dialog=dialogEnterValueInteger, Result=OK, NumpadKeypadSet=True
    Button (191,131 150x30), "Cancel"
        OnMouseClick: CloseDialog Dialog=dialogEnterValueInteger, Result=Cancel, NumpadKeypadSet=True
END_VISUALIZATION

// ---- HMI1/Screens/Dialogs/dialogReject.TcVIS
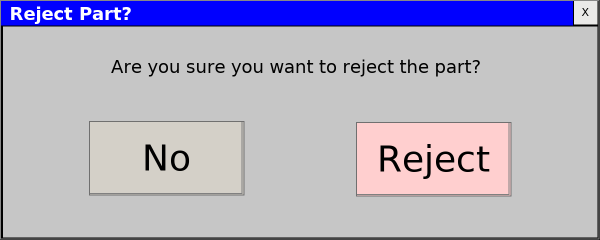
VISUALIZATION dialogReject  // 600x240
    Rectangle (0,0 600x240)
    Button (356,122 155x74), "Reject"
        OnMouseClick: CloseDialog Dialog=dialogReject, Result=Yes, NumpadKeypadSet=True
    Button (89,121 155x74), "No"
        OnMouseClick: CloseDialog Dialog=dialogReject, Result=No, NumpadKeypadSet=True
    Label (74,43 444x48), "Are you sure you want to reject the part?"
    Rectangle (0,0 600x26), "Reject Part?"
    Rectangle (573,0 25x25), "X"
        OnMouseClick: CloseDialog Dialog=dialogReject, Result=Cancel, NumpadKeypadSet=True
END_VISUALIZATION

// ---- HMI1/Screens/Dialogs/dialogDeviceInfo.TcVIS
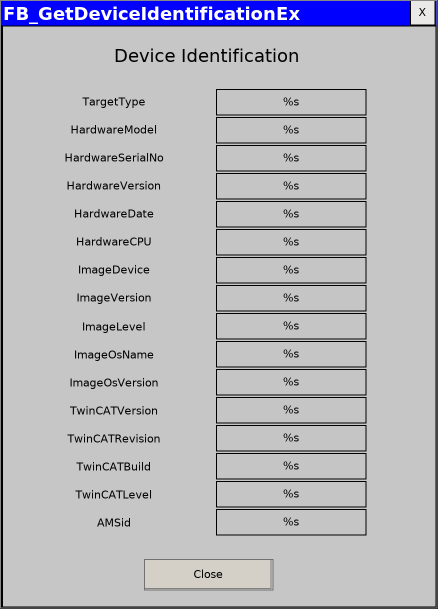
VISUALIZATION dialogDeviceInfo  // 438x609
    Rectangle (0,0 438x609)
        OnMouseClick: CloseDialog Dialog=dialogDeviceInfo, Result=OK, NumpadKeypadSet=True
    Button (144,559 129x31), "Close"
        OnMouseClick: CloseDialog Dialog=dialogDeviceInfo, Result=None, NumpadKeypadSet=True
    Rectangle (0,0 438x26), "FB_GetDeviceIdentificationEx"
    Rectangle (410,0 25x25), "X"
        OnMouseClick: CloseDialog Dialog=dialogDeviceInfo, Result=Cancel, NumpadKeypadSet=True
    Rectangle (216,89 150x26), "%s", text variable: System.sysDeviceInfo.strTargetType
    Label (16,89 196x26), "TargetType"
    Label (16,117 196x26), "HardwareModel"
    Rectangle (216,117 150x26), "%s", text variable: System.sysDeviceInfo.strHardwareModel
    Rectangle (216,145 150x26), "%s", text variable: System.sysDeviceInfo.strHardwareSerialNo
    Label (16,145 196x26), "HardwareSerialNo"
    Label (16,173 196x26), "HardwareVersion"
    Rectangle (216,173 150x26), "%s", text variable: System.sysDeviceInfo.strHardwareVersion
    Rectangle (216,201 150x26), "%s", text variable: System.sysDeviceInfo.strHardwareDate
    Label (16,201 196x26), "HardwareDate"
    Label (16,229 196x26), "HardwareCPU"
    Rectangle (216,229 150x26), "%s", text variable: System.sysDeviceInfo.strHardwareCPU
    Rectangle (216,257 150x26), "%s", text variable: System.sysDeviceInfo.strImageDevice
    Label (16,257 196x26), "ImageDevice"
    Label (16,285 196x26), "ImageVersion"
    Rectangle (216,285 150x26), "%s", text variable: System.sysDeviceInfo.strImageVersion
    Rectangle (216,313 150x26), "%s", text variable: System.sysDeviceInfo.strImageLevel
    Label (16,314 196x26), "ImageLevel"
    Label (16,342 196x26), "ImageOsName"
    Rectangle (216,341 150x26), "%s", text variable: System.sysDeviceInfo.strImageOsName
    Rectangle (216,369 150x26), "%s", text variable: System.sysDeviceInfo.strImageOsVersion
    Label (16,370 196x26), "ImageOsVersion"
    Label (16,398 196x26), "TwinCATVersion"
    Rectangle (216,397 150x26), "%s", text variable: System.sysDeviceInfo.strTwinCATVersion
    Rectangle (216,425 150x26), "%s", text variable: System.sysDeviceInfo.strTwinCATRevision
    Label (16,426 196x26), "TwinCATRevision"
    Rectangle (216,453 150x26), "%s", text variable: System.sysDeviceInfo.strTwinCATBuild
    Label (16,454 196x26), "TwinCATBuild"
    Label (16,482 196x26), "TwinCATLevel"
    Rectangle (216,481 150x26), "%s", text variable: System.sysDeviceInfo.strTwinCATLevel
    Label (16,510 196x26), "AMSid"
    Rectangle (216,509 150x26), "%s", text variable: System.sysDeviceInfo.strAmsNetId
    Label (109,43 196x26), "Device Identification"
END_VISUALIZATION

// ---- HMI1/Screens/Dialogs/dialogGetLicensesEx.TcVIS
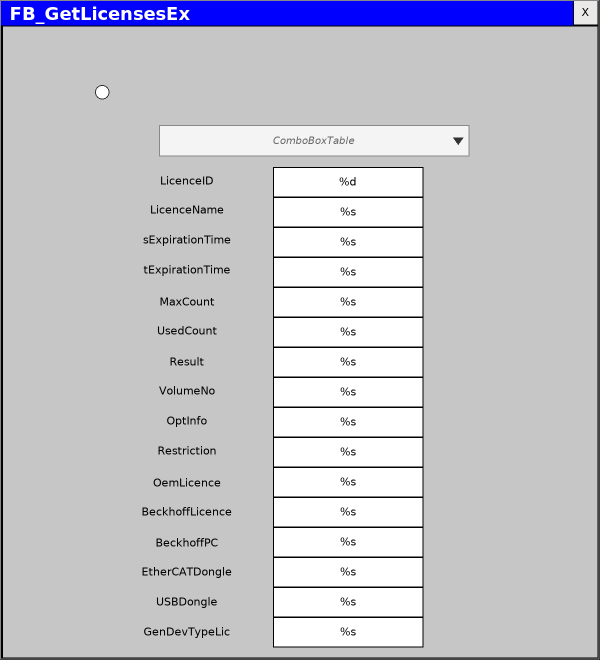
VISUALIZATION dialogGetLicensesEx  // 600x660
    Rectangle (0,0 600x660)
        OnMouseClick: CloseDialog Dialog=dialogGetLicensesEx, Result=OK, NumpadKeypadSet=True
    Rectangle (0,0 600x26), "FB_GetLicensesEx"
    Rectangle (573,0 25x25), "X"
        OnMouseClick: CloseDialog Dialog=dialogGetLicensesEx, Result=Cancel, NumpadKeypadSet=True
    Rectangle (273,167 150x30), "%d", text variable: gLicenceView.tActiveLicenceArray.stLicenseId
    Label (112,166 150x30), "LicenceID"
    Label (112,195 150x30), "LicenceName"
    Rectangle (273,197 150x30), "%s", text variable: gLicenceView.tActiveLicenceArray.sLicenseName
    Label (112,225 150x30), "sExpirationTime"
    Rectangle (273,227 150x30), "%s", text variable: gLicenceView.tActiveLicenceArray.sExpirationTime
    Label (112,255 150x30), "tExpirationTime"
    Rectangle (273,257 150x30), "%s"
    Label (112,287 150x30), "MaxCount"
    Rectangle (273,287 150x30), "%s", text variable: gLicenceView.tActiveLicenceArray.nMaxCount
    Label (112,316 150x30), "UsedCount"
    Rectangle (273,317 150x30), "%s", text variable: gLicenceView.tActiveLicenceArray.nUsedCount
    Rectangle (273,347 150x30), "%s", text variable: gLicenceView.tActiveLicenceArray.eResult
    Label (112,347 150x30), "Result"
    Label (112,376 150x30), "VolumeNo"
    Rectangle (273,377 150x30), "%s", text variable: gLicenceView.tActiveLicenceArray.nVolumeNo
    Label (112,406 150x30), "OptInfo"
    Rectangle (273,407 150x30), "%s", text variable: gLicenceView.tActiveLicenceArray.nOptInfo
    Label (112,436 150x30), "Restriction"
    Rectangle (273,437 150x30), "%s", text variable: gLicenceView.tActiveLicenceArray.nRestriction
    Label (112,468 150x30), "OemLicence"
    Rectangle (273,467 150x30), "%s", text variable: gLicenceView.tActiveLicenceArray.bOemLicense
    Label (112,497 150x30), "BeckhoffLicence"
    Rectangle (273,497 150x30), "%s", text variable: gLicenceView.tActiveLicenceArray.bBeckhoffLicense
    Rectangle (273,527 150x30), "%s", text variable: gLicenceView.tActiveLicenceArray.bBeckhoffPC
    Label (112,528 150x30), "BeckhoffPC"
    Label (112,557 150x30), "EtherCATDongle"
    Rectangle (273,557 150x30), "%s", text variable: gLicenceView.tActiveLicenceArray.bEtherCATDongle
    Label (112,587 150x30), "USBDongle"
    Rectangle (273,587 150x30), "%s", text variable: gLicenceView.tActiveLicenceArray.bUSBDongle
    Label (112,617 150x30), "GenDevTypeLic"
    Rectangle (273,617 150x30), "%s", text variable: gLicenceView.tActiveLicenceArray.bGenDevTypeLic
    RadioButton (93,37 454x110), variable: gLicenceView.licenceType
        Areas[0]: Text=Valid Licences
        Areas[1]: Text=Pending Licences
        Areas[2]: Text=Demo Licences
        Areas[3]: Text=OEM Licences
        Areas[4]: Text=Failed Licences
        Areas[5]: Text=Invalid Licences
    ComboBoxTable (159,125 310x31), variable: gLicenceView.tActiveLicenceSel, data array: gLicenceView.tActiveLicenceList
        p1892666644: System.tActiveLicenceArray.sLicenseName
        p338671338: System.tActiveLicenceArray.tExpirationTime
        p2170511999: System.tActiveLicenceArray.sExpirationTime
        p3723444502: System.tActiveLicenceArray.nMaxCount
        p1218418051: System.tActiveLicenceArray.nUsedCount
        p746581629: System.tActiveLicenceArray.eResult
        p3104783080: System.tActiveLicenceArray.nVolumeNo
        p2501879983: System.tActiveLicenceArray.nOptInfo
        p7306298: System.tActiveLicenceArray.nRestriction
        p1933151965: System.tActiveLicenceArray.bOemLicense
        p3863566920: System.tActiveLicenceArray.bBeckhoffLicense
        p2192122294: System.tActiveLicenceArray.bBeckhoffPC
        p400160035: System.tActiveLicenceArray.bEtherCATDongle
        p1265227338: System.tActiveLicenceArray.bUSBDongle
        p3726181087: System.tActiveLicenceArray.bGenDevTypeLic
        p3854506369: gLicenceView.tActiveLicenceList[INDEX]
END_VISUALIZATION

// ---- HMI1/Screens/Dialogs/dialogEnterValue.TcVIS
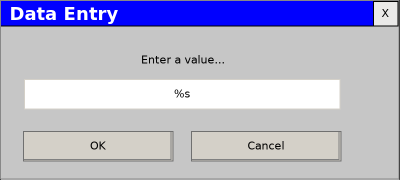
VISUALIZATION dialogEnterValue  // 400x180
VAR_IN_OUT
	enteredValue:STRING;
		
END_VAR
    Rectangle (0,0 400x188)
    Rectangle (0,0 400x26), "Data Entry"
    Rectangle (373,1 25x25), "X"
        OnMouseClick: CloseDialog Dialog=dialogEnterValue, Result=Cancel, NumpadKeypadSet=True
    Label (108,45 150x30), "Enter a value..."
    Textfield (24,79 316x30), "%s", text variable: enteredValue
        OnMouseClick: write enteredValue via VisuDialogs.Numpad
    Button (23,131 150x30), "OK"
        OnMouseClick: CloseDialog Dialog=dialogEnterValue, Result=OK, NumpadKeypadSet=True
    Button (191,131 150x30), "Cancel"
        OnMouseClick: CloseDialog Dialog=dialogEnterValue, Result=Cancel, NumpadKeypadSet=True
END_VISUALIZATION

// ---- HMI1/Screens/Dialogs/visuDataDisplay.TcVIS
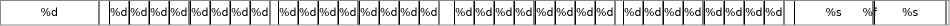
VISUALIZATION visuDataDisplay  // 950x26
VAR_IN_OUT
	d:dutDWord; //data for faceplate
END_VAR
    Rectangle (0,0 99x25), "%d", text variable: d.memLoc
    Rectangle (109,0 20x25), "%d", text variable: d.b38, colour toggle: d.b38, invisible if: d.Hideb3
    Rectangle (129,0 20x25), "%d", text variable: d.b37, colour toggle: d.b37, invisible if: d.Hideb3
    Rectangle (149,0 20x25), "%d", text variable: d.b36, colour toggle: d.b36, invisible if: d.Hideb3
    Rectangle (169,0 20x25), "%d", text variable: d.b35, colour toggle: d.b35, invisible if: d.Hideb3
    Rectangle (190,0 20x25), "%d", text variable: d.b34, colour toggle: d.b34, invisible if: d.Hideb3
    Rectangle (210,0 20x25), "%d", text variable: d.b33, colour toggle: d.b33, invisible if: d.Hideb3
    Rectangle (230,0 20x25), "%d", text variable: d.b32, colour toggle: d.b32, invisible if: d.Hideb3
    Rectangle (250,0 20x25), "%d", text variable: d.b31, colour toggle: d.b31, invisible if: d.Hideb3
    Rectangle (278,0 20x25), "%d", text variable: d.b28, colour toggle: d.b28, invisible if: d.Hideb2
    Rectangle (298,0 20x25), "%d", text variable: d.b27, colour toggle: d.b27, invisible if: d.Hideb2
    Rectangle (318,0 20x25), "%d", text variable: d.b26, colour toggle: d.b26, invisible if: d.Hideb2
    Rectangle (338,0 20x25), "%d", text variable: d.b25, colour toggle: d.b25, invisible if: d.Hideb2
    Rectangle (359,0 20x25), "%d", text variable: d.b24, colour toggle: d.b24, invisible if: d.Hideb2
    Rectangle (379,0 20x25), "%d", text variable: d.b23, colour toggle: d.b23, invisible if: d.Hideb2
    Rectangle (399,0 20x25), "%d", text variable: d.b22, colour toggle: d.b22, invisible if: d.Hideb2
    Rectangle (419,0 20x25), "%d", text variable: d.b21, colour toggle: d.b21, invisible if: d.Hideb2
    Rectangle (454,0 20x25), "%d", text variable: d.b18, colour toggle: d.b18, invisible if: d.Hideb1
    Rectangle (474,0 20x25), "%d", text variable: d.b17, colour toggle: d.b17, invisible if: d.Hideb1
    Rectangle (494,0 20x25), "%d", text variable: d.b16, colour toggle: d.b16, invisible if: d.Hideb1
    Rectangle (514,0 20x25), "%d", text variable: d.b15, colour toggle: d.b15, invisible if: d.Hideb1
    Rectangle (535,0 20x25), "%d", text variable: d.b14, colour toggle: d.b14, invisible if: d.Hideb1
    Rectangle (555,0 20x25), "%d", text variable: d.b13, colour toggle: d.b13, invisible if: d.Hideb1
    Rectangle (575,0 20x25), "%d", text variable: d.b12, colour toggle: d.b12, invisible if: d.Hideb1
    Rectangle (595,0 20x25), "%d", text variable: d.b11, colour toggle: d.b11, invisible if: d.Hideb1
    Rectangle (623,0 20x25), "%d", text variable: d.b08, colour toggle: d.b08, invisible if: d.Hideb0
    Rectangle (643,0 20x25), "%d", text variable: d.b07, colour toggle: d.b07, invisible if: d.Hideb0
    Rectangle (663,0 20x25), "%d", text variable: d.b06, colour toggle: d.b06, invisible if: d.Hideb0
    Rectangle (683,0 20x25), "%d", text variable: d.b05, colour toggle: d.b05, invisible if: d.Hideb0
    Rectangle (704,0 20x25), "%d", text variable: d.b04, colour toggle: d.b04, invisible if: d.Hideb0
    Rectangle (724,0 20x25), "%d", text variable: d.b03, colour toggle: d.b03, invisible if: d.Hideb0
    Rectangle (744,0 20x25), "%d", text variable: d.b02, colour toggle: d.b02, invisible if: d.Hideb0
    Rectangle (764,0 20x25), "%d", text variable: d.b01, colour toggle: d.b01, invisible if: d.Hideb0
    Rectangle (794,0 79x25), "%s", text variable: d.hexVal, invisible if: d.ShowREAL
    Rectangle (874,0 72x25), "%s", text variable: d.valStr, invisible if: d.ShowREAL
    Rectangle (794,0 152x25), "%f", text variable: d.floatVal, invisible if: d.ShowHex
END_VISUALIZATION

// ---- HMI1/Screens/Dialogs/visuTaskData.TcVIS
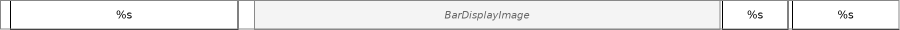
VISUALIZATION visuTaskData  // 900x30
VAR_IN_OUT
	d:typeIndividualTask; //data for faceplate
END_VAR
    Rectangle (10,0 228x30), "%s", text variable: d.singleTaskName, invisible if: NOT d.IsTaskEnabled
    BarDisplayImage (254,0 466x30), value: d.CycleTimeActual, invisible if: NOT d.IsTaskEnabled, style: BarDisplayImage-Gray, scale format: %.1f, scale 0..100
    Rectangle (792,0 107x30), "%s", invisible if: NOT d.IsTaskEnabled, text list: 'TaskText', text index: d.TaskStatus, colour variable: d.StateColour
    Rectangle (722,0 66x30), "%s", text variable: d.complexity, invisible if: NOT d.IsTaskEnabled, colour variable: d.StateColour
END_VISUALIZATION

// ---- HMI1/Screens/Layout/Lay_040_MachineLayout.TcVIS
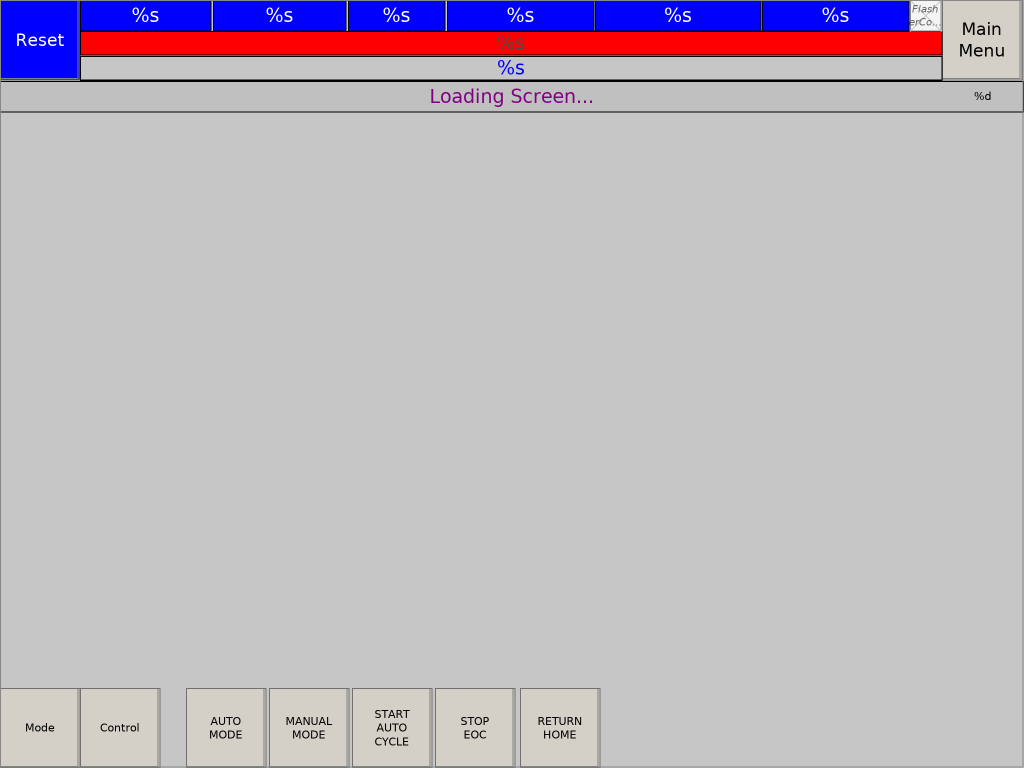
VISUALIZATION Lay_040_MachineLayout  // 1024x768
    Frame (0,0 1024x768)
        shows Tmp_000_Template(header := gHMIData.hmiHeader)
END_VISUALIZATION

// ---- HMI1/Screens/Machine Settings/MaS_800_SettingScreen.TcVIS
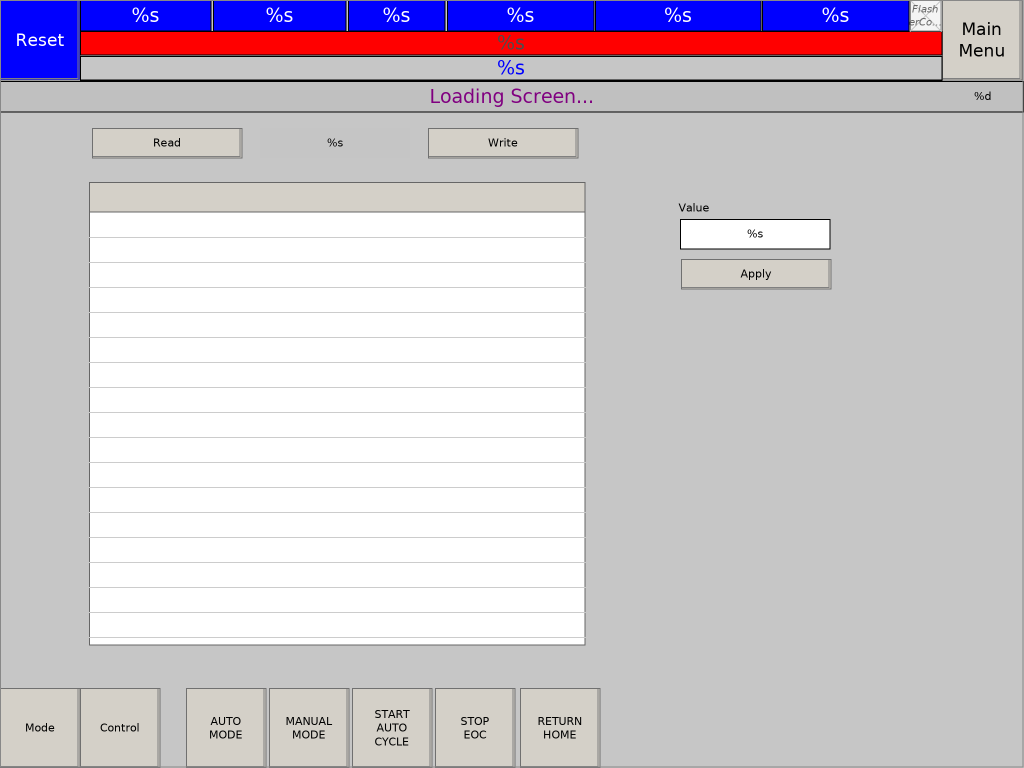
VISUALIZATION MaS_800_SettingScreen  // 1024x768
    Frame (0,0 1024x768)
        shows Tmp_000_Template(header := gHMIData.hmiHeader)
    Table (89,182 496x463), data array: MachineSettings.Setting
        p1420305297: MachineSettings.varSelectedColumn
        p4052804203: MachineSettings.varSelectedColumnValid
        p1137915858: MachineSettings.varSelectedRow
        p1822360349: MachineSettings.varSelectedRowValid
        p1128707560: MachineSettings.numElementsOfSettings
        p3854506369: MachineSettings.Setting[INDEX].TextName
        p1892666644: MachineSettings.Setting[INDEX].Value
        p338671338: MachineSettings.Setting[INDEX].hasChanged
        Columns.Column.[1].Template: OnMouseClick: execute { MachineSettings.numSelectedSettingNew := MachineSettings.Setting[MachineSettings.varSelectedRow].Value; }
    Button (92,128 150x30), "Read"
        tap MachineSettings.btnRead
        OnMouseDown: execute { gHMIButtons.gAnyButtonPressed := TRUE; }
    Button (428,128 150x30), "Write"
        tap MachineSettings.btnWrite
        OnMouseDown: execute { gHMIButtons.gAnyButtonPressed := TRUE; }
    Label (619,193 150x30), "Value"
    Rectangle (680,219 150x30), "%s", text variable: MachineSettings.numSelectedSettingNew
        OnMouseClick: OpenDialog Dialog=dialogEnterValueInteger, Parameters={enteredValue: MachineSettings.numSelectedSettingNew}, Selected={1: }, OpenModal=True, OpenCentered=True
    Button (681,259 150x30), "Apply"
        tap MachineSettings.btnMoveValue
        OnMouseDown: execute { gHMIButtons.gAnyButtonPressed := TRUE; }
    Rectangle (260,128 150x30), "%s", text variable: MachineSettings.strStatusFeeback, text list: ''
END_VISUALIZATION

// ---- HMI1/Screens/Menu/Men_030_MenuScreen.TcVIS
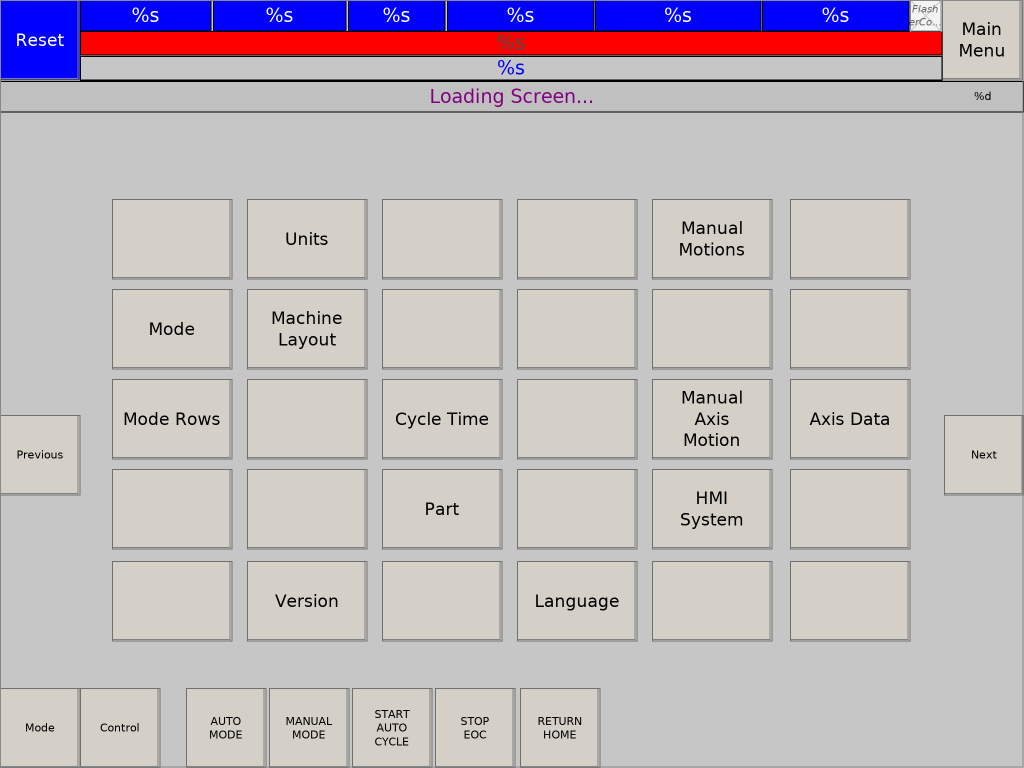
VISUALIZATION Men_030_MenuScreen  // 1024x768
    Frame (0,0 1024x768)
        shows Tmp_000_Template(header := gHMIData.hmiHeader)
    Button (112,199 120x80), text list: ''
        OnMouseDown: execute { gHMIButtons.gAnyButtonPressed := TRUE; }
    Button (247,199 120x80), "Units", text list: ''
        OnMouseDown: execute { gHMIButtons.gAnyButtonPressed := TRUE; }
        OnMouseDown: change screen: Unt_401_Units
    Button (382,199 120x80), text list: ''
        OnMouseDown: execute { gHMIButtons.gAnyButtonPressed := TRUE; }
    Button (517,199 120x80), text list: ''
        OnMouseDown: execute { gHMIButtons.gAnyButtonPressed := TRUE; }
    Button (652,199 120x80), "Manual Motions", text list: ''
        OnMouseClick: change screen: Mot_010_Motions
        OnMouseDown: execute { gHMIButtons.gAnyButtonPressed := TRUE; }
    Button (790,199 120x80), text list: ''
        OnMouseDown: execute { gHMIButtons.gAnyButtonPressed := TRUE; }
    Button (112,289 120x80), "Mode", text list: ''
        OnMouseDown: execute { gHMIButtons.gAnyButtonPressed := TRUE; }
        OnMouseDown: change screen: Mod_001_ModeScreen
    Button (247,289 120x80), "Machine Layout", text list: ''
        OnMouseDown: execute { gHMIButtons.gAnyButtonPressed := TRUE; }
        OnMouseDown: change screen: Lay_040_MachineLayout
    Button (382,289 120x80), text list: ''
        OnMouseDown: execute { gHMIButtons.gAnyButtonPressed := TRUE; }
    Button (517,289 120x80), text list: ''
        OnMouseDown: execute { gHMIButtons.gAnyButtonPressed := TRUE; }
    Button (652,289 120x80), text list: ''
        OnMouseDown: execute { gHMIButtons.gAnyButtonPressed := TRUE; }
    Button (790,289 120x80), text list: ''
        OnMouseDown: execute { gHMIButtons.gAnyButtonPressed := TRUE; }
    Button (112,379 120x80), "Mode Rows", text list: ''
        OnMouseDown: execute { gHMIButtons.gAnyButtonPressed := TRUE; }
        OnMouseDown: change screen: Mod_002_ModeScreenRows
    Button (247,379 120x80), text list: ''
        OnMouseDown: execute { gHMIButtons.gAnyButtonPressed := TRUE; }
    Button (382,379 120x80), "Cycle Time", text list: ''
        OnMouseDown: execute { gHMIButtons.gAnyButtonPressed := TRUE; }
        OnMouseDown: change screen: Prc_501_Cycle
    Button (517,379 120x80), text list: ''
        OnMouseDown: execute { gHMIButtons.gAnyButtonPressed := TRUE; }
    Button (652,379 120x80), "Manual Axis Motion", text list: ''
        OnMouseDown: execute { gHMIButtons.gAnyButtonPressed := TRUE; }
        OnMouseDown: change screen: Mot_011_Axis
    Button (790,379 120x80), "Axis Data", text list: ''
        OnMouseDown: execute { gHMIButtons.gAnyButtonPressed := TRUE; }
        OnMouseDown: change screen: Unt_402_Axis
    Button (112,469 120x80), text list: ''
        OnMouseDown: execute { gHMIButtons.gAnyButtonPressed := TRUE; }
    Button (247,469 120x80), text list: ''
        OnMouseDown: execute { gHMIButtons.gAnyButtonPressed := TRUE; }
    Button (382,469 120x80), "Part", text list: ''
        OnMouseDown: execute { gHMIButtons.gAnyButtonPressed := TRUE; }
        OnMouseDown: change screen: Prc_500_Part
    Button (517,469 120x80), text list: ''
        OnMouseDown: execute { gHMIButtons.gAnyButtonPressed := TRUE; }
    Button (652,469 120x80), "HMI System", text list: ''
        OnMouseDown: execute { gHMIButtons.gAnyButtonPressed := TRUE; }
        OnMouseDown: change screen: Sys_901_HMISystem
    Button (790,469 120x80), text list: ''
        OnMouseDown: execute { gHMIButtons.gAnyButtonPressed := TRUE; }
    Button (112,561 120x80), text list: ''
        OnMouseDown: execute { gHMIButtons.gAnyButtonPressed := TRUE; }
    Button (247,561 120x80), "Version", text list: ''
        OnMouseDown: execute { gHMIButtons.gAnyButtonPressed := TRUE; }
        OnMouseDown: change screen: Sys_902_Version
    Button (382,561 120x80), text list: ''
        OnMouseDown: execute { gHMIButtons.gAnyButtonPressed := TRUE; }
    Button (517,561 120x80), "Language", text list: ''
        OnMouseDown: execute { gHMIButtons.gAnyButtonPressed := TRUE; }
        OnMouseDown: change screen: Unt_403_Language
    Button (652,561 120x80), text list: ''
        OnMouseDown: execute { gHMIButtons.gAnyButtonPressed := TRUE; }
    Button (790,561 120x80), text list: ''
        OnMouseDown: execute { gHMIButtons.gAnyButtonPressed := TRUE; }
    Group (0,415 1024x80)
        Button (0,0 80x80), "Previous"
            OnMouseClick: change screen: Men_032_MenuScreen_3
            OnMouseDown: execute { gHMIButtons.gAnyButtonPressed := TRUE; }
        Button (944,0 80x80), "Next"
            OnMouseClick: change screen: Men_031_MenuScreen_2
            OnMouseDown: execute { gHMIButtons.gAnyButtonPressed := TRUE; }
END_VISUALIZATION

// ---- HMI1/Screens/Menu/Men_031_MenuScreen_2.TcVIS
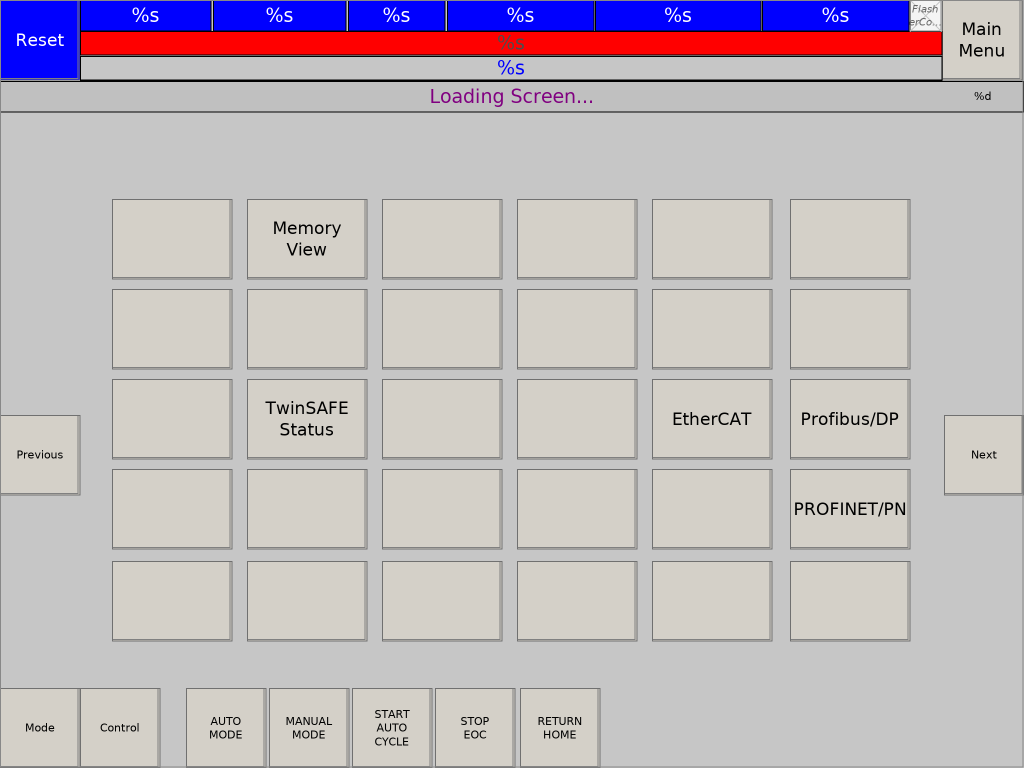
VISUALIZATION Men_031_MenuScreen_2  // 1024x768
    Frame (0,0 1024x768)
        shows Tmp_000_Template(header := gHMIData.hmiHeader)
    Button (112,199 120x80), text list: ''
        OnMouseDown: execute { gHMIButtons.gAnyButtonPressed := TRUE; }
    Button (247,199 120x80), "Memory View", text list: ''
        OnMouseClick: change screen: Dia_800_DataDisplay
        OnMouseDown: execute { gHMIButtons.gAnyButtonPressed := TRUE; }
    Button (382,199 120x80), text list: ''
        OnMouseDown: execute { gHMIButtons.gAnyButtonPressed := TRUE; }
    Button (517,199 120x80), text list: ''
        OnMouseDown: execute { gHMIButtons.gAnyButtonPressed := TRUE; }
    Button (652,199 120x80), text list: ''
        OnMouseDown: execute { gHMIButtons.gAnyButtonPressed := TRUE; }
    Button (790,199 120x80), text list: ''
        OnMouseDown: execute { gHMIButtons.gAnyButtonPressed := TRUE; }
    Button (112,289 120x80), text list: ''
        OnMouseDown: execute { gHMIButtons.gAnyButtonPressed := TRUE; }
    Button (247,289 120x80), text list: ''
        OnMouseDown: execute { gHMIButtons.gAnyButtonPressed := TRUE; }
    Button (382,289 120x80), text list: ''
        OnMouseDown: execute { gHMIButtons.gAnyButtonPressed := TRUE; }
    Button (517,289 120x80), text list: ''
        OnMouseDown: execute { gHMIButtons.gAnyButtonPressed := TRUE; }
    Button (652,289 120x80), text list: ''
        OnMouseDown: execute { gHMIButtons.gAnyButtonPressed := TRUE; }
    Button (790,289 120x80), text list: ''
        OnMouseDown: execute { gHMIButtons.gAnyButtonPressed := TRUE; }
    Button (112,379 120x80), text list: ''
        OnMouseDown: execute { gHMIButtons.gAnyButtonPressed := TRUE; }
    Button (247,379 120x80), "TwinSAFE Status", text list: ''
        OnMouseClick: change screen: Saf_700_SafetyStatus
        OnMouseDown: execute { gHMIButtons.gAnyButtonPressed := TRUE; }
    Button (382,379 120x80), text list: ''
        OnMouseDown: execute { gHMIButtons.gAnyButtonPressed := TRUE; }
    Button (517,379 120x80), text list: ''
        OnMouseDown: execute { gHMIButtons.gAnyButtonPressed := TRUE; }
    Button (652,379 120x80), "EtherCAT", text list: ''
        OnMouseClick: change screen: Dia_801_EtherCAT
        OnMouseDown: execute { gHMIButtons.gAnyButtonPressed := TRUE; }
    Button (790,379 120x80), "Profibus/DP", text list: ''
        OnMouseClick: change screen: Dia_802_Profibus
        OnMouseDown: execute { gHMIButtons.gAnyButtonPressed := TRUE; }
    Button (112,469 120x80), text list: ''
        OnMouseDown: execute { gHMIButtons.gAnyButtonPressed := TRUE; }
    Button (247,469 120x80), text list: ''
        OnMouseDown: execute { gHMIButtons.gAnyButtonPressed := TRUE; }
    Button (382,469 120x80), text list: ''
        OnMouseDown: execute { gHMIButtons.gAnyButtonPressed := TRUE; }
    Button (517,469 120x80), text list: ''
        OnMouseDown: execute { gHMIButtons.gAnyButtonPressed := TRUE; }
    Button (652,469 120x80), text list: ''
        OnMouseDown: execute { gHMIButtons.gAnyButtonPressed := TRUE; }
    Button (790,469 120x80), "PROFINET/PN", text list: ''
        OnMouseClick: change screen: Dia_803_ProfiNet
        OnMouseDown: execute { gHMIButtons.gAnyButtonPressed := TRUE; }
    Button (112,561 120x80), text list: ''
        OnMouseDown: execute { gHMIButtons.gAnyButtonPressed := TRUE; }
    Button (247,561 120x80), text list: ''
        OnMouseDown: execute { gHMIButtons.gAnyButtonPressed := TRUE; }
    Button (382,561 120x80), text list: ''
        OnMouseDown: execute { gHMIButtons.gAnyButtonPressed := TRUE; }
    Button (517,561 120x80), text list: ''
        OnMouseDown: execute { gHMIButtons.gAnyButtonPressed := TRUE; }
    Button (652,561 120x80), text list: ''
        OnMouseDown: execute { gHMIButtons.gAnyButtonPressed := TRUE; }
    Button (790,561 120x80), text list: ''
        OnMouseDown: execute { gHMIButtons.gAnyButtonPressed := TRUE; }
    Group (0,415 1024x80)
        Button (0,0 80x80), "Previous"
            OnMouseClick: change screen: Men_030_MenuScreen
            OnMouseDown: execute { gHMIButtons.gAnyButtonPressed := TRUE; }
        Button (944,0 80x80), "Next"
            OnMouseClick: change screen: Men_032_MenuScreen_3
            OnMouseDown: execute { gHMIButtons.gAnyButtonPressed := TRUE; }
END_VISUALIZATION

// ---- HMI1/Screens/Menu/Men_032_MenuScreen_3.TcVIS
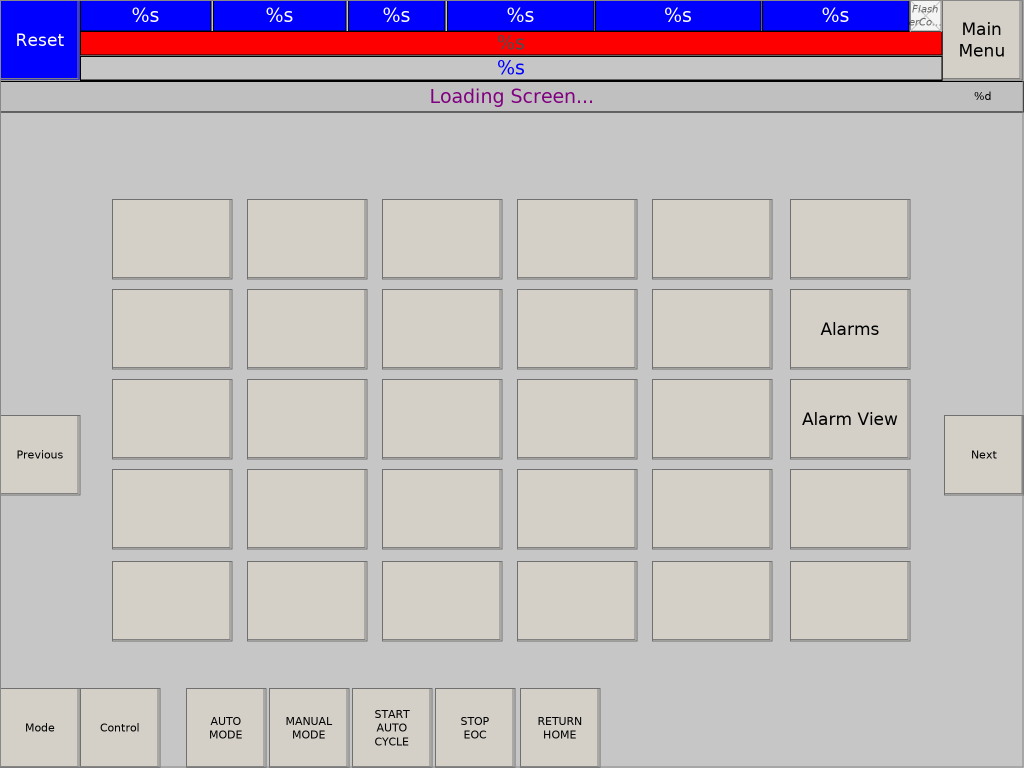
VISUALIZATION Men_032_MenuScreen_3  // 1024x768
    Frame (0,0 1024x768)
        shows Tmp_000_Template(header := gHMIData.hmiHeader)
    Group (0,415 1024x80)
        Button (0,0 80x80), "Previous"
            OnMouseClick: change screen: Men_031_MenuScreen_2
            OnMouseDown: execute { gHMIButtons.gAnyButtonPressed := TRUE; }
        Button (944,0 80x80), "Next"
            OnMouseClick: change screen: Men_030_MenuScreen
            OnMouseDown: execute { gHMIButtons.gAnyButtonPressed := TRUE; }
    Button (112,199 120x80), text list: ''
        OnMouseDown: execute { gHMIButtons.gAnyButtonPressed := TRUE; }
    Button (247,199 120x80), text list: ''
        OnMouseClick: change screen: Dia_800_DataDisplay
        OnMouseDown: execute { gHMIButtons.gAnyButtonPressed := TRUE; }
    Button (382,199 120x80), text list: ''
        OnMouseDown: execute { gHMIButtons.gAnyButtonPressed := TRUE; }
    Button (517,199 120x80), text list: ''
        OnMouseDown: execute { gHMIButtons.gAnyButtonPressed := TRUE; }
    Button (652,199 120x80), text list: ''
        OnMouseDown: execute { gHMIButtons.gAnyButtonPressed := TRUE; }
    Button (790,199 120x80), text list: ''
        OnMouseDown: execute { gHMIButtons.gAnyButtonPressed := TRUE; }
    Button (112,289 120x80), text list: ''
        OnMouseDown: execute { gHMIButtons.gAnyButtonPressed := TRUE; }
    Button (247,289 120x80), text list: ''
        OnMouseDown: execute { gHMIButtons.gAnyButtonPressed := TRUE; }
    Button (382,289 120x80), text list: ''
        OnMouseDown: execute { gHMIButtons.gAnyButtonPressed := TRUE; }
    Button (517,289 120x80), text list: ''
        OnMouseDown: execute { gHMIButtons.gAnyButtonPressed := TRUE; }
    Button (652,289 120x80), text list: ''
        OnMouseDown: execute { gHMIButtons.gAnyButtonPressed := TRUE; }
    Button (790,289 120x80), "Alarms", text list: ''
        OnMouseClick: change screen: Msg_020_Alarms
        OnMouseDown: execute { gHMIButtons.gAnyButtonPressed := TRUE; }
    Button (112,379 120x80), text list: ''
        OnMouseDown: execute { gHMIButtons.gAnyButtonPressed := TRUE; }
    Button (247,379 120x80), text list: ''
        OnMouseClick: change screen: Saf_700_SafetyStatus
        OnMouseDown: execute { gHMIButtons.gAnyButtonPressed := TRUE; }
    Button (382,379 120x80), text list: ''
        OnMouseDown: execute { gHMIButtons.gAnyButtonPressed := TRUE; }
    Button (517,379 120x80), text list: ''
        OnMouseDown: execute { gHMIButtons.gAnyButtonPressed := TRUE; }
    Button (652,379 120x80), text list: ''
        OnMouseClick: change screen: Dia_801_EtherCAT
        OnMouseDown: execute { gHMIButtons.gAnyButtonPressed := TRUE; }
    Button (790,379 120x80), "Alarm View", text list: ''
        OnMouseClick: change screen: Msg_021_AlarmsView
        OnMouseDown: execute { gHMIButtons.gAnyButtonPressed := TRUE; }
    Button (112,469 120x80), text list: ''
        OnMouseDown: execute { gHMIButtons.gAnyButtonPressed := TRUE; }
    Button (247,469 120x80), text list: ''
        OnMouseDown: execute { gHMIButtons.gAnyButtonPressed := TRUE; }
    Button (382,469 120x80), text list: ''
        OnMouseDown: execute { gHMIButtons.gAnyButtonPressed := TRUE; }
    Button (517,469 120x80), text list: ''
        OnMouseDown: execute { gHMIButtons.gAnyButtonPressed := TRUE; }
    Button (652,469 120x80), text list: ''
        OnMouseDown: execute { gHMIButtons.gAnyButtonPressed := TRUE; }
    Button (790,469 120x80), text list: ''
        OnMouseClick: change screen: Dia_803_ProfiNet
        OnMouseDown: execute { gHMIButtons.gAnyButtonPressed := TRUE; }
    Button (112,561 120x80), text list: ''
        OnMouseDown: execute { gHMIButtons.gAnyButtonPressed := TRUE; }
    Button (247,561 120x80), text list: ''
        OnMouseDown: execute { gHMIButtons.gAnyButtonPressed := TRUE; }
    Button (382,561 120x80), text list: ''
        OnMouseDown: execute { gHMIButtons.gAnyButtonPressed := TRUE; }
    Button (517,561 120x80), text list: ''
        OnMouseDown: execute { gHMIButtons.gAnyButtonPressed := TRUE; }
    Button (652,561 120x80), text list: ''
        OnMouseDown: execute { gHMIButtons.gAnyButtonPressed := TRUE; }
    Button (790,561 120x80), text list: ''
        OnMouseDown: execute { gHMIButtons.gAnyButtonPressed := TRUE; }
END_VISUALIZATION

// ---- HMI1/Screens/Messages/Msg_020_Alarms.TcVIS
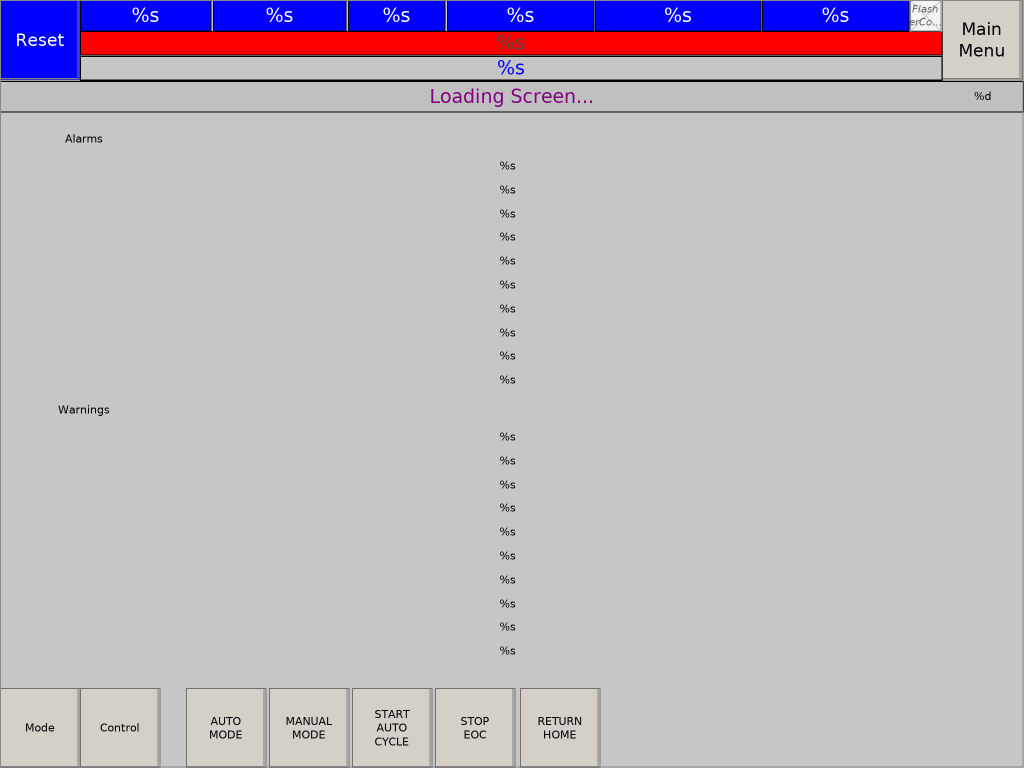
VISUALIZATION Msg_020_Alarms  // 1024x768
    Frame (0,0 1024x768)
        shows Tmp_000_Template(header := gHMIData.hmiHeader)
    Frame (0,152 1024x30)
        shows MessageRow(msg := gHMIData.gAlarmViewMsg.AlarmViewMsg[1])
    Frame (0,176 1024x30)
        shows MessageRow(msg := gHMIData.gAlarmViewMsg.AlarmViewMsg[2])
    Frame (0,200 1024x30)
        shows MessageRow(msg := gHMIData.gAlarmViewMsg.AlarmViewMsg[3])
    Frame (0,223 1024x30)
        shows MessageRow(msg := gHMIData.gAlarmViewMsg.AlarmViewMsg[4])
    Frame (0,247 1024x30)
        shows MessageRow(msg := gHMIData.gAlarmViewMsg.AlarmViewMsg[5])
    Frame (0,271 1024x30)
        shows MessageRow(msg := gHMIData.gAlarmViewMsg.AlarmViewMsg[6])
    Frame (0,295 1024x30)
        shows MessageRow(msg := gHMIData.gAlarmViewMsg.AlarmViewMsg[7])
    Frame (0,319 1024x30)
        shows MessageRow(msg := gHMIData.gAlarmViewMsg.AlarmViewMsg[8])
    Frame (0,342 1024x30)
        shows MessageRow(msg := gHMIData.gAlarmViewMsg.AlarmViewMsg[9])
    Rectangle (9,124 150x30), "Alarms"
    Frame (0,366 1024x30)
        shows MessageRow(msg := gHMIData.gAlarmViewMsg.AlarmViewMsg[10])
    Frame (0,423 1024x30)
        shows MessageRow(msg := gHMIData.gAlarmViewMsg.WarningViewMsg[1])
    Frame (0,447 1024x30)
        shows MessageRow(msg := gHMIData.gAlarmViewMsg.WarningViewMsg[2])
    Frame (0,471 1024x30)
        shows MessageRow(msg := gHMIData.gAlarmViewMsg.WarningViewMsg[3])
    Frame (0,494 1024x30)
        shows MessageRow(msg := gHMIData.gAlarmViewMsg.WarningViewMsg[4])
    Frame (0,518 1024x30)
        shows MessageRow(msg := gHMIData.gAlarmViewMsg.WarningViewMsg[5])
    Frame (0,542 1024x30)
        shows MessageRow(msg := gHMIData.gAlarmViewMsg.WarningViewMsg[6])
    Frame (0,566 1024x30)
        shows MessageRow(msg := gHMIData.gAlarmViewMsg.WarningViewMsg[7])
    Frame (0,590 1024x30)
        shows MessageRow(msg := gHMIData.gAlarmViewMsg.WarningViewMsg[8])
    Frame (0,613 1024x30)
        shows MessageRow(msg := gHMIData.gAlarmViewMsg.WarningViewMsg[9])
    Rectangle (9,395 150x30), "Warnings"
    Frame (0,637 1024x30)
        shows MessageRow(msg := gHMIData.gAlarmViewMsg.WarningViewMsg[10])
END_VISUALIZATION

// ---- HMI1/Screens/Messages/Msg_021_AlarmsView.TcVIS
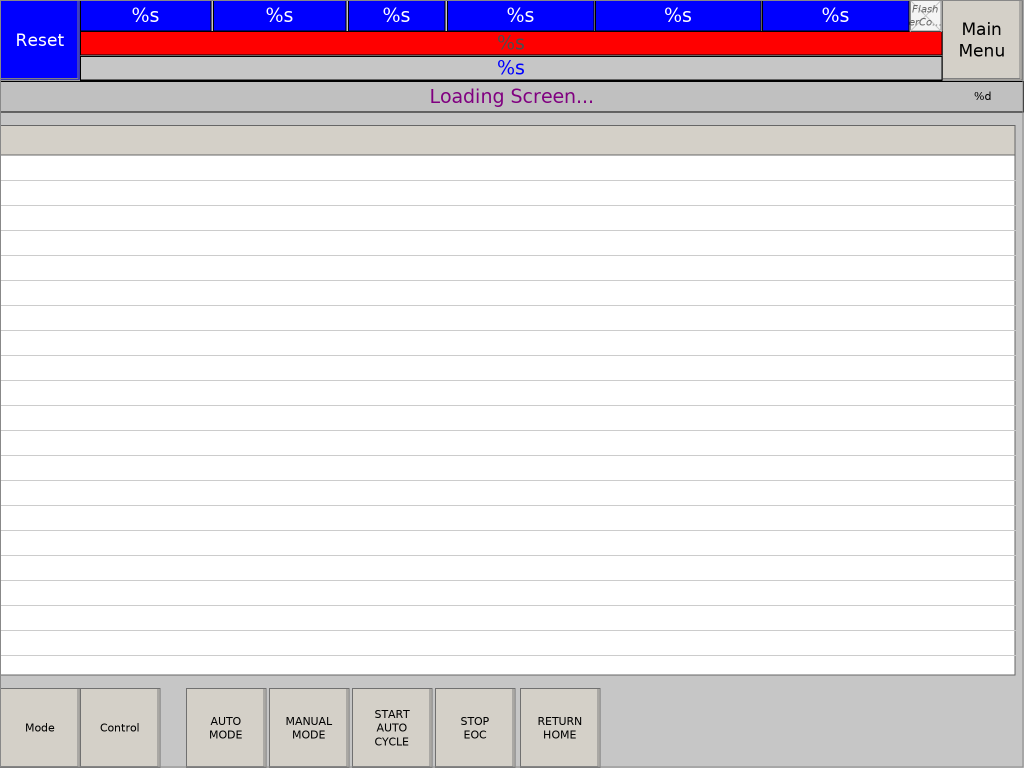
VISUALIZATION Msg_021_AlarmsView  // 1024x768
    Frame (0,0 1024x768)
        shows Tmp_000_Template(header := gHMIData.hmiHeader)
    Table (0,125 1015x550), data array: GlobalMessages.gHMIAlarmView.msgArry
        p3854506369: GlobalMessages.gHMIAlarmView.msgArry[INDEX].timeRaised
        p1892666644: GlobalMessages.gHMIAlarmView.msgArry[INDEX].text
        p338671338: GlobalMessages.gHMIAlarmView.msgArry[INDEX].timeResolved
        p2170511999: GlobalMessages.gHMIAlarmView.msgArry[INDEX].source
        p2232123230: Time Raised
        p511219082: Message Text
        p1755163831: Time Resolved
        p4092479075: Location
        Columns.Column.[0].Template: GlobalMessages.gHMIAlarmView.msgArryStyle[INDEX].isColoured; GlobalMessages.gHMIAlarmView.msgArryStyle[INDEX].colourToApply
        Columns.Column.[1].Template: GlobalMessages.gHMIAlarmView.msgArryStyle[INDEX].isColoured; GlobalMessages.gHMIAlarmView.msgArryStyle[INDEX].colourToApply
        Columns.Column.[2].Template: GlobalMessages.gHMIAlarmView.msgArryStyle[INDEX].isColoured; GlobalMessages.gHMIAlarmView.msgArryStyle[INDEX].colourToApply
        Columns.Column.[3].Template: GlobalMessages.gHMIAlarmView.msgArryStyle[INDEX].isColoured; GlobalMessages.gHMIAlarmView.msgArryStyle[INDEX].colourToApply
END_VISUALIZATION

// ---- HMI1/Screens/Mode/Mod_001_ModeScreen.TcVIS
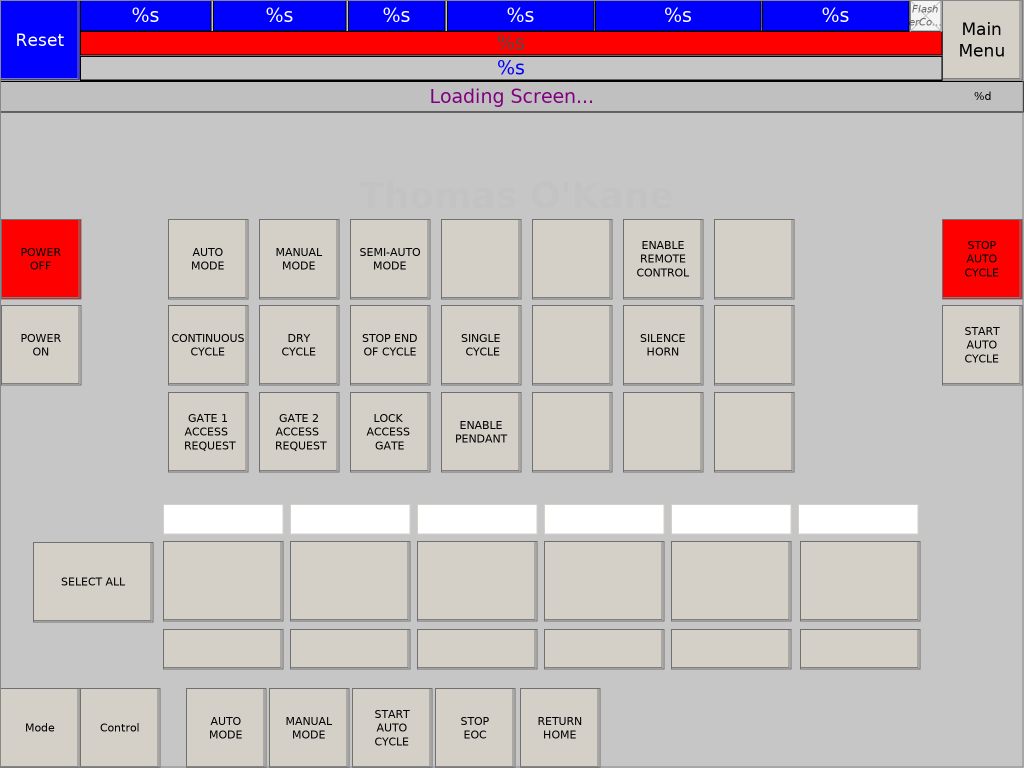
VISUALIZATION Mod_001_ModeScreen  // 1024x768
    Frame (0,0 1024x768)
        shows Tmp_000_Template(header := gHMIData.hmiHeader)
    Group (1,219 1021x166)
        Group (941,0 80x166)
            Button (0,0 80x80), "STOP AUTO CYCLE", text list: ''
                tap gHMIButtons.btnMode.btnAutoCycleStopPressed
                OnMouseDown: execute { gHMIButtons.gAnyButtonPressed := TRUE; }
            Button (0,86 80x80), "START AUTO CYCLE", colour toggle: gHMIButtons.btnFdbk.btnAutoCyclingFdbk, text list: ''
                tap gHMIButtons.btnMode.btnAutoCycleStartPressed
                OnMouseDown: execute { gHMIButtons.gAnyButtonPressed := TRUE; }
        Button (0,86 80x80), "POWER ON", colour toggle: Mc_Global.PowerOnFdbk, text list: ''
            tap gHMIButtons.btnMode.btnPowerOnPressed
            OnMouseDown: execute { gHMIButtons.gAnyButtonPressed := TRUE; }
        Button (0,0 80x80), "POWER OFF", text list: ''
            tap gHMIButtons.btnMode.btnPowerOffPressed
            OnMouseDown: execute { gHMIButtons.gAnyButtonPressed := TRUE; }
    Group (17,162 1000x310)
        Rectangle (0,0 1000x67), "Thomas O'Kane"
        Button (151,57 80x80), "AUTO MODE", colour toggle: gHMIButtons.btnFdbk.btn00Fdbk, invisible if: gHMIButtons.btnHides.btn00Hide, text list: ''
            tap gHMIButtons.btnMode.btn00Pressed
            OnMouseDown: execute { gHMIButtons.gAnyButtonPressed := TRUE; }
        Button (242,57 80x80), "MANUAL MODE", colour toggle: gHMIButtons.btnFdbk.btn01Fdbk, invisible if: gHMIButtons.btnHides.btn01Hide, text list: ''
            tap gHMIButtons.btnMode.btn01Pressed
            OnMouseDown: execute { gHMIButtons.gAnyButtonPressed := TRUE; }
        Button (333,57 80x80), "SEMI-AUTO MODE", colour toggle: gHMIButtons.btnFdbk.btn02Fdbk, invisible if: gHMIButtons.btnHides.btn02Hide, text list: ''
            tap gHMIButtons.btnMode.btn02Pressed
            OnMouseDown: execute { gHMIButtons.gAnyButtonPressed := TRUE; }
        Button (424,57 80x80), colour toggle: gHMIButtons.btnFdbk.btn03Fdbk, invisible if: gHMIButtons.btnHides.btn03Hide, text list: ''
            tap gHMIButtons.btnMode.btn03Pressed
            OnMouseDown: execute { gHMIButtons.gAnyButtonPressed := TRUE; }
        Button (606,57 80x80), "ENABLE REMOTE CONTROL", colour toggle: gHMIButtons.btnFdbk.btn05Fdbk, invisible if: gHMIButtons.btnHides.btn05Hide, text list: ''
            tap gHMIButtons.btnMode.btn05Pressed
            OnMouseDown: execute { gHMIButtons.gAnyButtonPressed := TRUE; }
        Button (515,57 80x80), colour toggle: gHMIButtons.btnFdbk.btn04Fdbk, invisible if: gHMIButtons.btnHides.btn04Hide, text list: ''
            tap gHMIButtons.btnMode.btn04Pressed
            OnMouseDown: execute { gHMIButtons.gAnyButtonPressed := TRUE; }
        Button (151,143 80x80), "CONTINUOUS CYCLE", colour toggle: gHMIButtons.btnFdbk.btn10Fdbk, invisible if: gHMIButtons.btnHides.btn10Hide, text list: ''
            tap gHMIButtons.btnMode.btn10Pressed
            OnMouseDown: execute { gHMIButtons.gAnyButtonPressed := TRUE; }
        Button (242,143 80x80), "DRY CYCLE", colour toggle: gHMIButtons.btnFdbk.btn11Fdbk, invisible if: gHMIButtons.btnHides.btn11Hide, text list: ''
            tap gHMIButtons.btnMode.btn11Pressed
            OnMouseDown: execute { gHMIButtons.gAnyButtonPressed := TRUE; }
        Button (333,143 80x80), "STOP END OF CYCLE", colour toggle: gHMIButtons.btnFdbk.btn12Fdbk, invisible if: gHMIButtons.btnHides.btn12Hide, text list: ''
            tap gHMIButtons.btnMode.btn12Pressed
            OnMouseDown: execute { gHMIButtons.gAnyButtonPressed := TRUE; }
        Button (424,143 80x80), "SINGLE CYCLE", colour toggle: gHMIButtons.btnFdbk.btn13Fdbk, invisible if: gHMIButtons.btnHides.btn13Hide, text list: ''
            tap gHMIButtons.btnMode.btn13Pressed
            OnMouseDown: execute { gHMIButtons.gAnyButtonPressed := TRUE; }
        Button (606,143 80x80), "SILENCE HORN", colour toggle: gHMIButtons.btnFdbk.btn15Fdbk, invisible if: gHMIButtons.btnHides.btn15Hide, text list: ''
            tap gHMIButtons.btnMode.btn15Pressed
            OnMouseDown: execute { gHMIButtons.gAnyButtonPressed := TRUE; }
        Button (515,143 80x80), colour toggle: gHMIButtons.btnFdbk.btn14Fdbk, invisible if: gHMIButtons.btnHides.btn14Hide, text list: ''
            tap gHMIButtons.btnMode.btn14Pressed
            OnMouseDown: execute { gHMIButtons.gAnyButtonPressed := TRUE; }
        Button (151,230 80x80), "GATE 1 ACCESS REQUEST", colour toggle: gHMIButtons.btnFdbk.btn20Fdbk, invisible if: gHMIButtons.btnHides.btn20Hide, text list: ''
            tap gHMIButtons.btnMode.btn20Pressed
            OnMouseDown: execute { gHMIButtons.gAnyButtonPressed := TRUE; }
        Button (242,230 80x80), "GATE 2 ACCESS REQUEST", colour toggle: gHMIButtons.btnFdbk.btn21Fdbk, invisible if: gHMIButtons.btnHides.btn21Hide, text list: ''
            tap gHMIButtons.btnMode.btn21Pressed
            OnMouseDown: execute { gHMIButtons.gAnyButtonPressed := TRUE; }
        Button (333,230 80x80), "LOCK ACCESS GATE", colour toggle: gHMIButtons.btnFdbk.btn22Fdbk, invisible if: gHMIButtons.btnHides.btn22Hide, text list: ''
            tap gHMIButtons.btnMode.btn22Pressed
            OnMouseDown: execute { gHMIButtons.gAnyButtonPressed := TRUE; }
        Button (424,230 80x80), "ENABLE PENDANT", colour toggle: gHMIButtons.btnFdbk.btn23Fdbk, invisible if: gHMIButtons.btnHides.btn23Hide, text list: ''
            tap gHMIButtons.btnMode.btn23Pressed
            OnMouseDown: execute { gHMIButtons.gAnyButtonPressed := TRUE; }
        Button (606,230 80x80), colour toggle: gHMIButtons.btnFdbk.btn25Fdbk, invisible if: gHMIButtons.btnHides.btn25Hide, text list: ''
            tap gHMIButtons.btnMode.btn25Pressed
            OnMouseDown: execute { gHMIButtons.gAnyButtonPressed := TRUE; }
        Button (515,230 80x80), colour toggle: gHMIButtons.btnFdbk.btn24Fdbk, invisible if: gHMIButtons.btnHides.btn24Hide, text list: ''
            tap gHMIButtons.btnMode.btn24Pressed
            OnMouseDown: execute { gHMIButtons.gAnyButtonPressed := TRUE; }
        Button (697,57 80x80), colour toggle: gHMIButtons.btnFdbk.btn06Fdbk, invisible if: gHMIButtons.btnHides.btn06Hide, text list: ''
            tap gHMIButtons.btnMode.btn06Pressed
            OnMouseDown: execute { gHMIButtons.gAnyButtonPressed := TRUE; }
        Button (697,143 80x80), colour toggle: gHMIButtons.btnFdbk.btn16Fdbk, invisible if: gHMIButtons.btnHides.btn16Hide, text list: ''
            tap gHMIButtons.btnMode.btn16Pressed
            OnMouseDown: execute { gHMIButtons.gAnyButtonPressed := TRUE; }
        Button (697,230 80x80), colour toggle: gHMIButtons.btnFdbk.btn26Fdbk, invisible if: gHMIButtons.btnHides.btn26Hide, text list: ''
            tap gHMIButtons.btnMode.btn26Pressed
            OnMouseDown: execute { gHMIButtons.gAnyButtonPressed := TRUE; }
    Textfield (163,504 120x30), invisible if: NOT gHMIData.gStationEnabled[1], text list: 'ModeStates', text index: S1_Global.station.Data.StationState, colour variable: S1_Global.station.Data.StationStateColour
        p55702900: S1_Global.station.Data.StationStateTextColour
    Textfield (290,504 120x30), invisible if: NOT gHMIData.gStationEnabled[2], text list: 'ModeStates', text index: S2_Global.station.Data.StationState, colour variable: S2_Global.station.Data.StationStateColour
        p55702900: S2_Global.station.Data.StationStateTextColour
    Textfield (417,504 120x30), invisible if: NOT gHMIData.gStationEnabled[3], text list: 'ModeStates', text index: S3_Global.station.Data.StationState, colour variable: S3_Global.station.Data.StationStateColour
        p55702900: S3_Global.station.Data.StationStateTextColour
    Textfield (544,504 120x30), invisible if: NOT gHMIData.gStationEnabled[4], text list: 'ModeStates', text index: S4_Global.station.Data.StationState, colour variable: S4_Global.station.Data.StationStateColour
        p55702900: S4_Global.station.Data.StationStateTextColour
    Textfield (671,504 120x30), invisible if: NOT gHMIData.gStationEnabled[5], text list: 'ModeStates', text index: S5_Global.station.Data.StationState, colour variable: S5_Global.station.Data.StationStateColour
        p55702900: S5_Global.station.Data.StationStateTextColour
    Textfield (798,504 120x30), invisible if: NOT gHMIData.gStationEnabled[6], text list: 'ModeStates', text index: S6_Global.station.Data.StationState, colour variable: S6_Global.station.Data.StationStateColour
        p55702900: S6_Global.station.Data.StationStateTextColour
    Button (163,541 120x80), colour toggle: gHMIData.gStationSelected[1], invisible if: NOT gHMIData.gStationEnabled[1], text list: 'StationNames', text index: 1
        tap gHMIButtons.btnSelectStation1
        OnMouseClick: execute { gHMIButtons.gAnyButtonPressed := TRUE; }
    Button (290,541 120x80), colour toggle: gHMIData.gStationSelected[2], invisible if: NOT gHMIData.gStationEnabled[2], text list: 'StationNames', text index: 2
        tap gHMIButtons.btnSelectStation2
        OnMouseClick: execute { gHMIButtons.gAnyButtonPressed := TRUE; }
    Button (417,541 120x80), colour toggle: gHMIData.gStationSelected[3], invisible if: NOT gHMIData.gStationEnabled[3], text list: 'StationNames', text index: 3
        tap gHMIButtons.btnSelectStation3
        OnMouseClick: execute { gHMIButtons.gAnyButtonPressed := TRUE; }
    Button (544,541 120x80), colour toggle: gHMIData.gStationSelected[4], invisible if: NOT gHMIData.gStationEnabled[4], text list: 'StationNames', text index: 4
        tap gHMIButtons.btnSelectStation4
        OnMouseClick: execute { gHMIButtons.gAnyButtonPressed := TRUE; }
    Button (671,541 120x80), colour toggle: gHMIData.gStationSelected[5], invisible if: NOT gHMIData.gStationEnabled[5], text list: 'StationNames', text index: 5
        tap gHMIButtons.btnSelectStation5
        OnMouseClick: execute { gHMIButtons.gAnyButtonPressed := TRUE; }
    Button (800,541 120x80), colour toggle: gHMIData.gStationSelected[6], invisible if: NOT gHMIData.gStationEnabled[6], text list: 'StationNames', text index: 6
        tap gHMIButtons.btnSelectStation6
        OnMouseClick: execute { gHMIButtons.gAnyButtonPressed := TRUE; }
    Button (33,542 120x80), "SELECT ALL", colour toggle: gHMIButtons.btnAllStationsSelected, text list: ''
        tap gHMIButtons.btnSelectAll
    Button (163,629 120x40), invisible if: NOT gHMIData.gStationEnabled[1], text list: 'stationLinked', text index: gHMIData.gStateLockStation1
        toggle gHMIButtons.btnLockStation1
        OnMouseClick: execute { gHMIButtons.gAnyButtonPressed := TRUE; }
    Button (290,629 120x40), invisible if: NOT gHMIData.gStationEnabled[2], text list: 'stationLinked', text index: gHMIData.gStateLockStation2
        toggle gHMIButtons.btnLockStation2
        OnMouseClick: execute { gHMIButtons.gAnyButtonPressed := TRUE; }
    Button (417,629 120x40), invisible if: NOT gHMIData.gStationEnabled[3], text list: 'stationLinked', text index: gHMIData.gStateLockStation3
        toggle gHMIButtons.btnLockStation3
        OnMouseClick: execute { gHMIButtons.gAnyButtonPressed := TRUE; }
    Button (544,629 120x40), invisible if: NOT gHMIData.gStationEnabled[4], text list: 'stationLinked', text index: gHMIData.gStateLockStation4
        toggle gHMIButtons.btnLockStation4
        OnMouseClick: execute { gHMIButtons.gAnyButtonPressed := TRUE; }
    Button (671,629 120x40), invisible if: NOT gHMIData.gStationEnabled[5], text list: 'stationLinked', text index: gHMIData.gStateLockStation5
        toggle gHMIButtons.btnLockStation5
        OnMouseClick: execute { gHMIButtons.gAnyButtonPressed := TRUE; }
    Button (800,629 120x40), invisible if: NOT gHMIData.gStationEnabled[6], text list: 'stationLinked', text index: gHMIData.gStateLockStation6
        toggle gHMIButtons.btnLockStation6
        OnMouseClick: execute { gHMIButtons.gAnyButtonPressed := TRUE; }
END_VISUALIZATION

// ---- HMI1/Screens/Mode/Mod_101_ModeScreen_Alternate.TcVIS
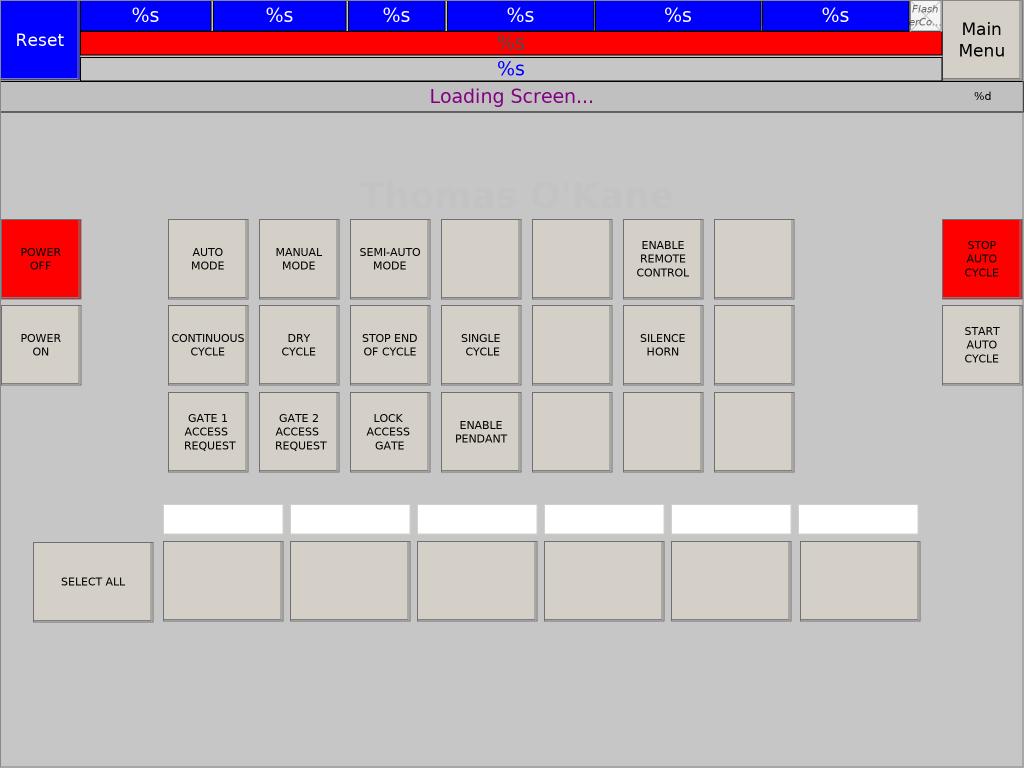
VISUALIZATION Mod_101_ModeScreen_Alternate  // 1024x768
    Frame (0,0 1024x768)
        shows Tmp_001_Template_Alternate(header := gHMIData.hmiHeader)
    Group (1,219 1021x166)
        Group (941,0 80x166)
            Button (0,0 80x80), "STOP AUTO CYCLE", text list: ''
                tap gHMIButtons.btnMode.btnAutoCycleStopPressed
                OnMouseDown: execute { gHMIButtons.gAnyButtonPressed := TRUE; }
            Button (0,86 80x80), "START AUTO CYCLE", colour toggle: gHMIButtons.btnFdbk.btnAutoCyclingFdbk, text list: ''
                tap gHMIButtons.btnMode.btnAutoCycleStartPressed
                OnMouseDown: execute { gHMIButtons.gAnyButtonPressed := TRUE; }
        Button (0,86 80x80), "POWER ON", colour toggle: Mc_Global.PowerOnFdbk, text list: ''
            tap gHMIButtons.btnMode.btnPowerOnPressed
            OnMouseDown: execute { gHMIButtons.gAnyButtonPressed := TRUE; }
        Button (0,0 80x80), "POWER OFF", text list: ''
            tap gHMIButtons.btnMode.btnPowerOffPressed
            OnMouseDown: execute { gHMIButtons.gAnyButtonPressed := TRUE; }
    Group (17,162 1000x310)
        Rectangle (0,0 1000x67), "Thomas O'Kane"
        Button (151,57 80x80), "AUTO MODE", colour toggle: gHMIButtons.btnFdbk.btn00Fdbk, invisible if: gHMIButtons.btnHides.btn00Hide, text list: ''
            tap gHMIButtons.btnMode.btn00Pressed
            OnMouseDown: execute { gHMIButtons.gAnyButtonPressed := TRUE; }
        Button (242,57 80x80), "MANUAL MODE", colour toggle: gHMIButtons.btnFdbk.btn01Fdbk, invisible if: gHMIButtons.btnHides.btn01Hide, text list: ''
            tap gHMIButtons.btnMode.btn01Pressed
            OnMouseDown: execute { gHMIButtons.gAnyButtonPressed := TRUE; }
        Button (333,57 80x80), "SEMI-AUTO MODE", colour toggle: gHMIButtons.btnFdbk.btn02Fdbk, invisible if: gHMIButtons.btnHides.btn02Hide, text list: ''
            tap gHMIButtons.btnMode.btn02Pressed
            OnMouseDown: execute { gHMIButtons.gAnyButtonPressed := TRUE; }
        Button (424,57 80x80), colour toggle: gHMIButtons.btnFdbk.btn03Fdbk, invisible if: gHMIButtons.btnHides.btn03Hide, text list: ''
            tap gHMIButtons.btnMode.btn03Pressed
            OnMouseDown: execute { gHMIButtons.gAnyButtonPressed := TRUE; }
        Button (606,57 80x80), "ENABLE REMOTE CONTROL", colour toggle: gHMIButtons.btnFdbk.btn05Fdbk, invisible if: gHMIButtons.btnHides.btn05Hide, text list: ''
            tap gHMIButtons.btnMode.btn05Pressed
            OnMouseDown: execute { gHMIButtons.gAnyButtonPressed := TRUE; }
        Button (515,57 80x80), colour toggle: gHMIButtons.btnFdbk.btn04Fdbk, invisible if: gHMIButtons.btnHides.btn04Hide, text list: ''
            tap gHMIButtons.btnMode.btn04Pressed
            OnMouseDown: execute { gHMIButtons.gAnyButtonPressed := TRUE; }
        Button (151,143 80x80), "CONTINUOUS CYCLE", colour toggle: gHMIButtons.btnFdbk.btn10Fdbk, invisible if: gHMIButtons.btnHides.btn10Hide, text list: ''
            tap gHMIButtons.btnMode.btn10Pressed
            OnMouseDown: execute { gHMIButtons.gAnyButtonPressed := TRUE; }
        Button (242,143 80x80), "DRY CYCLE", colour toggle: gHMIButtons.btnFdbk.btn11Fdbk, invisible if: gHMIButtons.btnHides.btn11Hide, text list: ''
            tap gHMIButtons.btnMode.btn11Pressed
            OnMouseDown: execute { gHMIButtons.gAnyButtonPressed := TRUE; }
        Button (333,143 80x80), "STOP END OF CYCLE", colour toggle: gHMIButtons.btnFdbk.btn12Fdbk, invisible if: gHMIButtons.btnHides.btn12Hide, text list: ''
            tap gHMIButtons.btnMode.btn12Pressed
            OnMouseDown: execute { gHMIButtons.gAnyButtonPressed := TRUE; }
        Button (424,143 80x80), "SINGLE CYCLE", colour toggle: gHMIButtons.btnFdbk.btn13Fdbk, invisible if: gHMIButtons.btnHides.btn13Hide, text list: ''
            tap gHMIButtons.btnMode.btn13Pressed
            OnMouseDown: execute { gHMIButtons.gAnyButtonPressed := TRUE; }
        Button (606,143 80x80), "SILENCE HORN", colour toggle: gHMIButtons.btnFdbk.btn15Fdbk, invisible if: gHMIButtons.btnHides.btn15Hide, text list: ''
            tap gHMIButtons.btnMode.btn15Pressed
            OnMouseDown: execute { gHMIButtons.gAnyButtonPressed := TRUE; }
        Button (515,143 80x80), colour toggle: gHMIButtons.btnFdbk.btn14Fdbk, invisible if: gHMIButtons.btnHides.btn14Hide, text list: ''
            tap gHMIButtons.btnMode.btn14Pressed
            OnMouseDown: execute { gHMIButtons.gAnyButtonPressed := TRUE; }
        Button (151,230 80x80), "GATE 1 ACCESS REQUEST", colour toggle: gHMIButtons.btnFdbk.btn20Fdbk, invisible if: gHMIButtons.btnHides.btn20Hide, text list: ''
            tap gHMIButtons.btnMode.btn20Pressed
            OnMouseDown: execute { gHMIButtons.gAnyButtonPressed := TRUE; }
        Button (242,230 80x80), "GATE 2 ACCESS REQUEST", colour toggle: gHMIButtons.btnFdbk.btn21Fdbk, invisible if: gHMIButtons.btnHides.btn21Hide, text list: ''
            tap gHMIButtons.btnMode.btn21Pressed
            OnMouseDown: execute { gHMIButtons.gAnyButtonPressed := TRUE; }
        Button (333,230 80x80), "LOCK ACCESS GATE", colour toggle: gHMIButtons.btnFdbk.btn22Fdbk, invisible if: gHMIButtons.btnHides.btn22Hide, text list: ''
            tap gHMIButtons.btnMode.btn22Pressed
            OnMouseDown: execute { gHMIButtons.gAnyButtonPressed := TRUE; }
        Button (424,230 80x80), "ENABLE PENDANT", colour toggle: gHMIButtons.btnFdbk.btn23Fdbk, invisible if: gHMIButtons.btnHides.btn23Hide, text list: ''
            tap gHMIButtons.btnMode.btn23Pressed
            OnMouseDown: execute { gHMIButtons.gAnyButtonPressed := TRUE; }
        Button (606,230 80x80), colour toggle: gHMIButtons.btnFdbk.btn25Fdbk, invisible if: gHMIButtons.btnHides.btn25Hide, text list: ''
            tap gHMIButtons.btnMode.btn25Pressed
            OnMouseDown: execute { gHMIButtons.gAnyButtonPressed := TRUE; }
        Button (515,230 80x80), colour toggle: gHMIButtons.btnFdbk.btn24Fdbk, invisible if: gHMIButtons.btnHides.btn24Hide, text list: ''
            tap gHMIButtons.btnMode.btn24Pressed
            OnMouseDown: execute { gHMIButtons.gAnyButtonPressed := TRUE; }
        Button (697,57 80x80), colour toggle: gHMIButtons.btnFdbk.btn06Fdbk, invisible if: gHMIButtons.btnHides.btn06Hide, text list: ''
            tap gHMIButtons.btnMode.btn06Pressed
            OnMouseDown: execute { gHMIButtons.gAnyButtonPressed := TRUE; }
        Button (697,143 80x80), colour toggle: gHMIButtons.btnFdbk.btn16Fdbk, invisible if: gHMIButtons.btnHides.btn16Hide, text list: ''
            tap gHMIButtons.btnMode.btn16Pressed
            OnMouseDown: execute { gHMIButtons.gAnyButtonPressed := TRUE; }
        Button (697,230 80x80), colour toggle: gHMIButtons.btnFdbk.btn26Fdbk, invisible if: gHMIButtons.btnHides.btn26Hide, text list: ''
            tap gHMIButtons.btnMode.btn26Pressed
            OnMouseDown: execute { gHMIButtons.gAnyButtonPressed := TRUE; }
    Group (33,504 887x118)
        Textfield (130,0 120x30), invisible if: NOT gHMIData.gStationEnabled[1], text list: 'ModeStates', text index: S1_Global.station.Data.StationState, colour variable: S1_Global.station.Data.StationStateColour
            p55702900: S1_Global.station.Data.StationStateTextColour
        Textfield (257,0 120x30), invisible if: NOT gHMIData.gStationEnabled[2], text list: 'ModeStates', text index: S2_Global.station.Data.StationState, colour variable: S2_Global.station.Data.StationStateColour
            p55702900: S2_Global.station.Data.StationStateTextColour
        Textfield (384,0 120x30), invisible if: NOT gHMIData.gStationEnabled[3], text list: 'ModeStates', text index: S3_Global.station.Data.StationState, colour variable: S3_Global.station.Data.StationStateColour
            p55702900: S3_Global.station.Data.StationStateTextColour
        Textfield (511,0 120x30), invisible if: NOT gHMIData.gStationEnabled[4], text list: 'ModeStates', text index: S4_Global.station.Data.StationState, colour variable: S4_Global.station.Data.StationStateColour
            p55702900: S4_Global.station.Data.StationStateTextColour
        Textfield (638,0 120x30), invisible if: NOT gHMIData.gStationEnabled[5], text list: 'ModeStates', text index: S5_Global.station.Data.StationState, colour variable: S5_Global.station.Data.StationStateColour
            p55702900: S5_Global.station.Data.StationStateTextColour
        Textfield (765,0 120x30), invisible if: NOT gHMIData.gStationEnabled[6], text list: 'ModeStates', text index: S6_Global.station.Data.StationState, colour variable: S6_Global.station.Data.StationStateColour
            p55702900: S6_Global.station.Data.StationStateTextColour
        Button (130,37 120x80), colour toggle: gHMIData.gStationSelected[1], invisible if: NOT gHMIData.gStationEnabled[1], text list: 'StationNames', text index: 1
            tap gHMIButtons.btnSelectStation1
        Button (257,37 120x80), colour toggle: gHMIData.gStationSelected[2], invisible if: NOT gHMIData.gStationEnabled[2], text list: 'StationNames', text index: 2
            tap gHMIButtons.btnSelectStation2
        Button (384,37 120x80), colour toggle: gHMIData.gStationSelected[3], invisible if: NOT gHMIData.gStationEnabled[3], text list: 'StationNames', text index: 3
            tap gHMIButtons.btnSelectStation3
        Button (511,37 120x80), colour toggle: gHMIData.gStationSelected[4], invisible if: NOT gHMIData.gStationEnabled[4], text list: 'StationNames', text index: 4
            tap gHMIButtons.btnSelectStation4
        Button (638,37 120x80), colour toggle: gHMIData.gStationSelected[5], invisible if: NOT gHMIData.gStationEnabled[5], text list: 'StationNames', text index: 5
            tap gHMIButtons.btnSelectStation5
        Button (767,37 120x80), colour toggle: gHMIData.gStationSelected[6], invisible if: NOT gHMIData.gStationEnabled[6], text list: 'StationNames', text index: 6
            tap gHMIButtons.btnSelectStation6
        Button (0,38 120x80), "SELECT ALL", colour toggle: gHMIButtons.btnAllStationsSelected, text list: ''
            tap gHMIButtons.btnSelectAll
END_VISUALIZATION

// ---- HMI1/Screens/Mode/Mod_002_ModeScreenRows.TcVIS
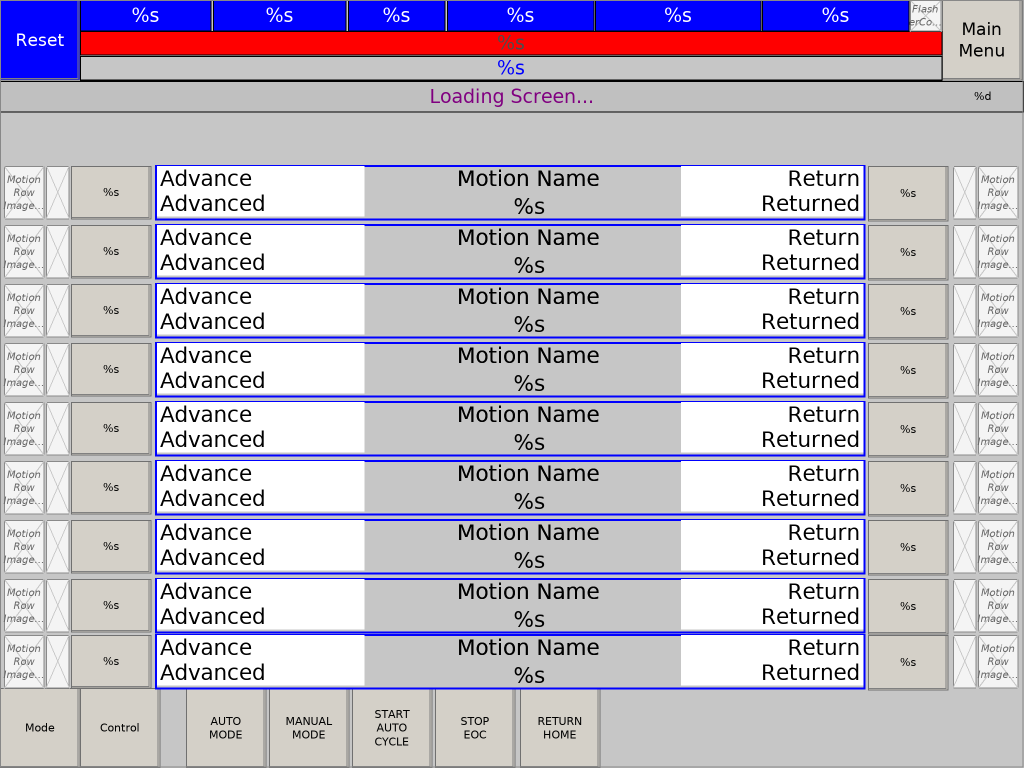
VISUALIZATION Mod_002_ModeScreenRows  // 1024x768
    Frame (0,0 1024x768)
        shows Tmp_000_Template(header := gHMIData.hmiHeader)
    Frame (0,165 1024x55)
        shows ModeRow(MotionRowInstanceSingle := gModeAlternate.gModeRows.gMotionRow1, MotionRowButtonsSingle := gModeAlternate.gModeButtons.gMotionRow1btn)
    Frame (0,224 1024x55)
        shows ModeRow(MotionRowInstanceSingle := gModeAlternate.gModeRows.gMotionRow2, MotionRowButtonsSingle := gModeAlternate.gModeButtons.gMotionRow2btn)
    Frame (0,283 1024x55)
        shows ModeRow(MotionRowInstanceSingle := gModeAlternate.gModeRows.gMotionRow3, MotionRowButtonsSingle := gModeAlternate.gModeButtons.gMotionRow3btn)
    Frame (0,342 1024x55)
        shows ModeRow(MotionRowInstanceSingle := gModeAlternate.gModeRows.gMotionRow4, MotionRowButtonsSingle := gModeAlternate.gModeButtons.gMotionRow4btn)
    Frame (0,401 1024x55)
        shows ModeRow(MotionRowInstanceSingle := gModeAlternate.gModeRows.gMotionRow5, MotionRowButtonsSingle := gModeAlternate.gModeButtons.gMotionRow5btn)
    Frame (0,460 1024x55)
        shows ModeRow(MotionRowInstanceSingle := gModeAlternate.gModeRows.gMotionRow6, MotionRowButtonsSingle := gModeAlternate.gModeButtons.gMotionRow6btn)
    Frame (0,519 1024x55)
        shows ModeRow(MotionRowInstanceSingle := gModeAlternate.gModeRows.gMotionRow7, MotionRowButtonsSingle := gModeAlternate.gModeButtons.gMotionRow7btn)
    Frame (0,578 1024x55)
        shows ModeRow(MotionRowInstanceSingle := gModeAlternate.gModeRows.gMotionRow8, MotionRowButtonsSingle := gModeAlternate.gModeButtons.gMotionRow8btn)
    Frame (0,634 1024x55)
        shows ModeRow(MotionRowInstanceSingle := gModeAlternate.gModeRows.gMotionRow9, MotionRowButtonsSingle := gModeAlternate.gModeButtons.gMotionRow9btn)
END_VISUALIZATION

